KUKA KRL program: demo_posicionaCubos.src, demo_posicionaCubos.dat

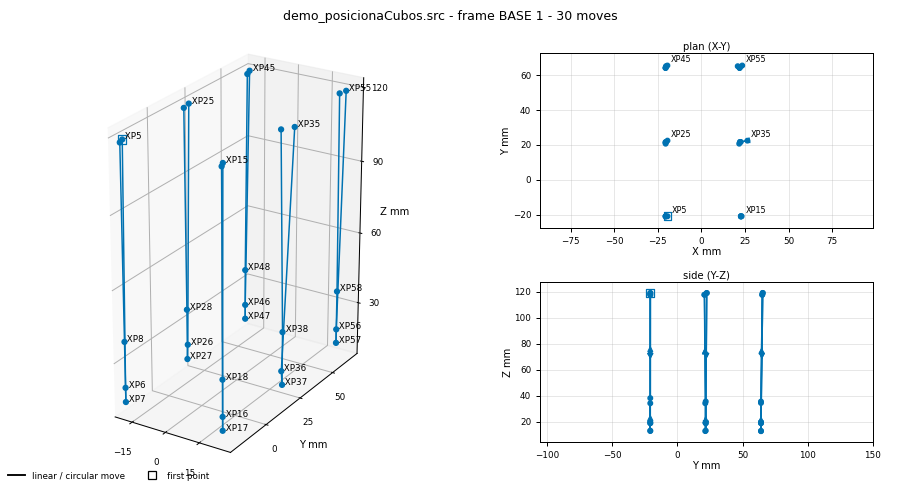
[picture p0: tool path of demo_posicionaCubos.src in frame BASE 1, 30 of 61 moves have a stored position in this frame; points joined in program order, loops and branches not executed]
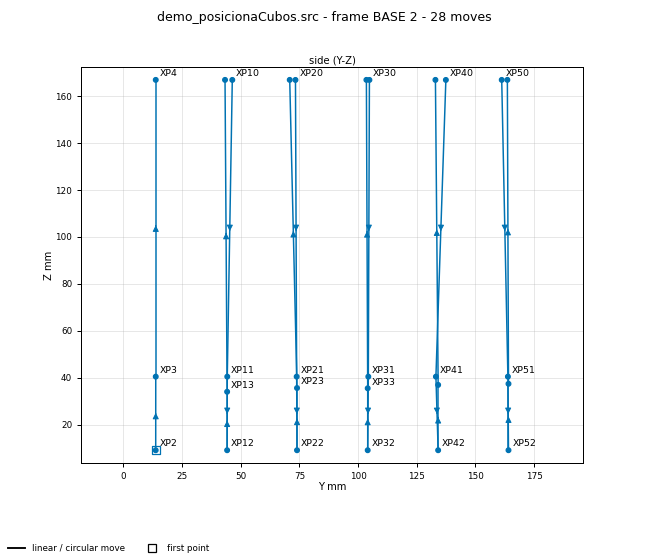
[picture p1: tool path of demo_posicionaCubos.src in frame BASE 2, 28 of 61 moves have a stored position in this frame; points joined in program order, loops and branches not executed]
--- demo_posicionaCubos.src ---
&ACCESS RVO1
&REL 186
&PARAM EDITMASK = *
&PARAM TEMPLATE = C:\KRC\Roboter\Template\vorgabe
DEF demo_posicionaCubos( )
;FOLD INI;%{PE}
  ;FOLD BASISTECH INI
    GLOBAL INTERRUPT DECL 3 WHEN $STOPMESS==TRUE DO IR_STOPM ( )
    INTERRUPT ON 3
    BAS (#INITMOV,0 )
  ;ENDFOLD (BASISTECH INI)
;FOLD SPOTTECH INI
USERSPOT(#INIT)
;ENDFOLD (SPOTTECH INI)
;FOLD GRIPPERTECH INI
USER_GRP(0,DUMMY,DUMMY,GDEFAULT)
;ENDFOLD (GRIPPERTECH INI)
  ;FOLD USER INI
    ;Make your modifications here

  ;ENDFOLD (USER INI)
;ENDFOLD (INI)
;FOLD SET GRIPPER_DEFAULT State=OPN CONT at START Delay=0 ms;%{PE}%R 8.3.1,%MKUKATPGRP,%CGRP,%VGRP,%P 2:1, 4:1, 5:#YES, 6:GDAT0, 8:0, 10:0
TRIGGER WHEN DISTANCE=0 DELAY=0 DO H50(GRP_APO,1,1,GCONT) PRIO=-1
;ENDFOLD
;FOLD PTP HOME  Vel= 100 % DEFAULT;%{PE}%MKUKATPBASIS,%CMOVE,%VPTP,%P 1:PTP, 2:HOME, 3:, 5:100, 7:DEFAULT
$BWDSTART = FALSE
PDAT_ACT=PDEFAULT
FDAT_ACT=FHOME
BAS (#PTP_PARAMS,100 )
$H_POS=XHOME
PTP  XHOME
;ENDFOLD
;FOLD PTP P1 CONT Vel=100 % PDAT2 Tool[1]:Gripper Base[0];%{PE}%R 8.3.34,%MKUKATPBASIS,%CMOVE,%VPTP,%P 1:PTP, 2:P1, 3:C_DIS, 5:100, 7:PDAT2
$BWDSTART=FALSE
PDAT_ACT=PPDAT2
FDAT_ACT=FP1
BAS(#PTP_PARAMS,100)
PTP XP1 C_DIS
;ENDFOLD
;FOLD LIN P2 CONT Vel=0.2 m/s CPDAT53 Tool[1]:Gripper Base[2]:cube_holder;%{PE}%R 8.3.34,%MKUKATPBASIS,%CMOVE,%VLIN,%P 1:LIN, 2:P2, 3:C_DIS C_DIS, 5:0.2, 7:CPDAT53
$BWDSTART=FALSE
LDAT_ACT=LCPDAT53
FDAT_ACT=FP2
BAS(#CP_PARAMS,0.2)
LIN XP2 C_DIS C_DIS
;ENDFOLD
;FOLD SET GRIPPER_DEFAULT State=CLO GDAT1;%{PE}%R 8.3.1,%MKUKATPGRP,%CGRP,%VGRP,%P 2:1, 4:2, 5:#NO, 6:GDAT1, 8:0, 10:0
H50(GRP,1,2,GGDAT1)
;ENDFOLD
;FOLD LIN P3 CONT Vel=0.2 m/s CPDAT54 Tool[1]:Gripper Base[2]:cube_holder;%{PE}%R 8.3.34,%MKUKATPBASIS,%CMOVE,%VLIN,%P 1:LIN, 2:P3, 3:C_DIS C_DIS, 5:0.2, 7:CPDAT54
$BWDSTART=FALSE
LDAT_ACT=LCPDAT54
FDAT_ACT=FP3
BAS(#CP_PARAMS,0.2)
LIN XP3 C_DIS C_DIS
;ENDFOLD
;FOLD LIN P4 CONT Vel=0.5 m/s CPDAT61 Tool[1]:Gripper Base[2]:cube_holder;%{PE}%R 8.3.34,%MKUKATPBASIS,%CMOVE,%VLIN,%P 1:LIN, 2:P4, 3:C_DIS C_DIS, 5:0.5, 7:CPDAT61
$BWDSTART=FALSE
LDAT_ACT=LCPDAT61
FDAT_ACT=FP4
BAS(#CP_PARAMS,0.5)
LIN XP4 C_DIS C_DIS
;ENDFOLD
;FOLD PTP P5 CONT Vel=80 % PDAT18 Tool[1]:Gripper Base[1]:verde;%{PE}%R 8.3.34,%MKUKATPBASIS,%CMOVE,%VPTP,%P 1:PTP, 2:P5, 3:C_DIS, 5:80, 7:PDAT18
$BWDSTART=FALSE
PDAT_ACT=PPDAT18
FDAT_ACT=FP5
BAS(#PTP_PARAMS,80)
PTP XP5 C_DIS
;ENDFOLD
;FOLD LIN P6 CONT Vel=0.5 m/s CPDAT57 Tool[1]:Gripper Base[1]:verde;%{PE}%R 8.3.34,%MKUKATPBASIS,%CMOVE,%VLIN,%P 1:LIN, 2:P6, 3:C_DIS C_DIS, 5:0.5, 7:CPDAT57
$BWDSTART=FALSE
LDAT_ACT=LCPDAT57
FDAT_ACT=FP6
BAS(#CP_PARAMS,0.5)
LIN XP6 C_DIS C_DIS
;ENDFOLD
;FOLD LIN P7 CONT Vel=0.2 m/s CPDAT58 Tool[1]:Gripper Base[1]:verde;%{PE}%R 8.3.34,%MKUKATPBASIS,%CMOVE,%VLIN,%P 1:LIN, 2:P7, 3:C_DIS C_DIS, 5:0.2, 7:CPDAT58
$BWDSTART=FALSE
LDAT_ACT=LCPDAT58
FDAT_ACT=FP7
BAS(#CP_PARAMS,0.2)
LIN XP7 C_DIS C_DIS
;ENDFOLD
;FOLD SET GRIPPER_DEFAULT State=OPN GDAT14;%{PE}%R 8.3.1,%MKUKATPGRP,%CGRP,%VGRP,%P 2:1, 4:1, 5:#NO, 6:GDAT14, 8:0, 10:0
H50(GRP,1,1,GGDAT14)
;ENDFOLD
;FOLD LIN P8 CONT Vel=0.2 m/s CPDAT59 Tool[1]:Gripper Base[1]:verde;%{PE}%R 8.3.34,%MKUKATPBASIS,%CMOVE,%VLIN,%P 1:LIN, 2:P8, 3:C_DIS C_DIS, 5:0.2, 7:CPDAT59
$BWDSTART=FALSE
LDAT_ACT=LCPDAT59
FDAT_ACT=FP8
BAS(#CP_PARAMS,0.2)
LIN XP8 C_DIS C_DIS
;ENDFOLD
;FOLD LIN P9 CONT Vel=0.5 m/s CPDAT60 Tool[1]:Gripper Base[1]:verde;%{PE}%R 8.3.34,%MKUKATPBASIS,%CMOVE,%VLIN,%P 1:LIN, 2:P9, 3:C_DIS C_DIS, 5:0.5, 7:CPDAT60
$BWDSTART=FALSE
LDAT_ACT=LCPDAT60
FDAT_ACT=FP9
BAS(#CP_PARAMS,0.5)
LIN XP9 C_DIS C_DIS
;ENDFOLD
;FOLD PTP P10 CONT Vel=80 % PDAT19 Tool[1]:Gripper Base[2]:cube_holder;%{PE}%R 8.3.34,%MKUKATPBASIS,%CMOVE,%VPTP,%P 1:PTP, 2:P10, 3:C_DIS, 5:80, 7:PDAT19
$BWDSTART=FALSE
PDAT_ACT=PPDAT19
FDAT_ACT=FP10
BAS(#PTP_PARAMS,80)
PTP XP10 C_DIS
;ENDFOLD
;FOLD LIN P11 CONT Vel=0.5 m/s CPDAT62 Tool[1]:Gripper Base[2]:cube_holder;%{PE}%R 8.3.34,%MKUKATPBASIS,%CMOVE,%VLIN,%P 1:LIN, 2:P11, 3:C_DIS C_DIS, 5:0.5, 7:CPDAT62
$BWDSTART=FALSE
LDAT_ACT=LCPDAT62
FDAT_ACT=FP11
BAS(#CP_PARAMS,0.5)
LIN XP11 C_DIS C_DIS
;ENDFOLD
;FOLD LIN P12 CONT Vel=0.2 m/s CPDAT63 Tool[1]:Gripper Base[2]:cube_holder;%{PE}%R 8.3.34,%MKUKATPBASIS,%CMOVE,%VLIN,%P 1:LIN, 2:P12, 3:C_DIS C_DIS, 5:0.2, 7:CPDAT63
$BWDSTART=FALSE
LDAT_ACT=LCPDAT63
FDAT_ACT=FP12
BAS(#CP_PARAMS,0.2)
LIN XP12 C_DIS C_DIS
;ENDFOLD
;FOLD SET GRIPPER_DEFAULT State=CLO GDAT15;%{PE}%R 8.3.1,%MKUKATPGRP,%CGRP,%VGRP,%P 2:1, 4:2, 5:#NO, 6:GDAT15, 8:0, 10:0
H50(GRP,1,2,GGDAT15)
;ENDFOLD
;FOLD LIN P13 CONT Vel=0.2 m/s CPDAT64 Tool[1]:Gripper Base[2]:cube_holder;%{PE}%R 8.3.34,%MKUKATPBASIS,%CMOVE,%VLIN,%P 1:LIN, 2:P13, 3:C_DIS C_DIS, 5:0.2, 7:CPDAT64
$BWDSTART=FALSE
LDAT_ACT=LCPDAT64
FDAT_ACT=FP13
BAS(#CP_PARAMS,0.2)
LIN XP13 C_DIS C_DIS
;ENDFOLD
;FOLD LIN P14 CONT Vel=0.5 m/s CPDAT65 Tool[1]:Gripper Base[2]:cube_holder;%{PE}%R 8.3.34,%MKUKATPBASIS,%CMOVE,%VLIN,%P 1:LIN, 2:P14, 3:C_DIS C_DIS, 5:0.5, 7:CPDAT65
$BWDSTART=FALSE
LDAT_ACT=LCPDAT65
FDAT_ACT=FP14
BAS(#CP_PARAMS,0.5)
LIN XP14 C_DIS C_DIS
;ENDFOLD
;FOLD PTP P15 CONT Vel=80 % PDAT20 Tool[1]:Gripper Base[1]:verde;%{PE}%R 8.3.34,%MKUKATPBASIS,%CMOVE,%VPTP,%P 1:PTP, 2:P15, 3:C_DIS, 5:80, 7:PDAT20
$BWDSTART=FALSE
PDAT_ACT=PPDAT20
FDAT_ACT=FP15
BAS(#PTP_PARAMS,80)
PTP XP15 C_DIS
;ENDFOLD
;FOLD LIN P16 CONT Vel=0.5 m/s CPDAT66 Tool[1]:Gripper Base[1]:verde;%{PE}%R 8.3.34,%MKUKATPBASIS,%CMOVE,%VLIN,%P 1:LIN, 2:P16, 3:C_DIS C_DIS, 5:0.5, 7:CPDAT66
$BWDSTART=FALSE
LDAT_ACT=LCPDAT66
FDAT_ACT=FP16
BAS(#CP_PARAMS,0.5)
LIN XP16 C_DIS C_DIS
;ENDFOLD
;FOLD LIN P17 CONT Vel=0.2 m/s CPDAT67 Tool[1]:Gripper Base[1]:verde;%{PE}%R 8.3.34,%MKUKATPBASIS,%CMOVE,%VLIN,%P 1:LIN, 2:P17, 3:C_DIS C_DIS, 5:0.2, 7:CPDAT67
$BWDSTART=FALSE
LDAT_ACT=LCPDAT67
FDAT_ACT=FP17
BAS(#CP_PARAMS,0.2)
LIN XP17 C_DIS C_DIS
;ENDFOLD
;FOLD SET GRIPPER_DEFAULT State=OPN GDAT16;%{PE}%R 8.3.1,%MKUKATPGRP,%CGRP,%VGRP,%P 2:1, 4:1, 5:#NO, 6:GDAT16, 8:0, 10:0
H50(GRP,1,1,GGDAT16)
;ENDFOLD
;FOLD LIN P18 CONT Vel=0.2 m/s CPDAT69 Tool[1]:Gripper Base[1]:verde;%{PE}%R 8.3.34,%MKUKATPBASIS,%CMOVE,%VLIN,%P 1:LIN, 2:P18, 3:C_DIS C_DIS, 5:0.2, 7:CPDAT69
$BWDSTART=FALSE
LDAT_ACT=LCPDAT69
FDAT_ACT=FP18
BAS(#CP_PARAMS,0.2)
LIN XP18 C_DIS C_DIS
;ENDFOLD
;FOLD LIN P19 CONT Vel=0.5 m/s CPDAT70 Tool[1]:Gripper Base[1]:verde;%{PE}%R 8.3.34,%MKUKATPBASIS,%CMOVE,%VLIN,%P 1:LIN, 2:P19, 3:C_DIS C_DIS, 5:0.5, 7:CPDAT70
$BWDSTART=FALSE
LDAT_ACT=LCPDAT70
FDAT_ACT=FP19
BAS(#CP_PARAMS,0.5)
LIN XP19 C_DIS C_DIS
;ENDFOLD
;FOLD PTP P20 CONT Vel=80 % PDAT21 Tool[1]:Gripper Base[2]:cube_holder;%{PE}%R 8.3.34,%MKUKATPBASIS,%CMOVE,%VPTP,%P 1:PTP, 2:P20, 3:C_DIS, 5:80, 7:PDAT21
$BWDSTART=FALSE
PDAT_ACT=PPDAT21
FDAT_ACT=FP20
BAS(#PTP_PARAMS,80)
PTP XP20 C_DIS
;ENDFOLD
;FOLD LIN P21 CONT Vel=0.5 m/s CPDAT71 Tool[1]:Gripper Base[2]:cube_holder;%{PE}%R 8.3.34,%MKUKATPBASIS,%CMOVE,%VLIN,%P 1:LIN, 2:P21, 3:C_DIS C_DIS, 5:0.5, 7:CPDAT71
$BWDSTART=FALSE
LDAT_ACT=LCPDAT71
FDAT_ACT=FP21
BAS(#CP_PARAMS,0.5)
LIN XP21 C_DIS C_DIS
;ENDFOLD
;FOLD LIN P22 CONT Vel=0.2 m/s CPDAT72 Tool[1]:Gripper Base[2]:cube_holder;%{PE}%R 8.3.34,%MKUKATPBASIS,%CMOVE,%VLIN,%P 1:LIN, 2:P22, 3:C_DIS C_DIS, 5:0.2, 7:CPDAT72
$BWDSTART=FALSE
LDAT_ACT=LCPDAT72
FDAT_ACT=FP22
BAS(#CP_PARAMS,0.2)
LIN XP22 C_DIS C_DIS
;ENDFOLD
;FOLD SET GRIPPER_DEFAULT State=CLO GDAT17;%{PE}%R 8.3.1,%MKUKATPGRP,%CGRP,%VGRP,%P 2:1, 4:2, 5:#NO, 6:GDAT17, 8:0, 10:0
H50(GRP,1,2,GGDAT17)
;ENDFOLD
;FOLD LIN P23 CONT Vel=0.2 m/s CPDAT73 Tool[1]:Gripper Base[2]:cube_holder;%{PE}%R 8.3.34,%MKUKATPBASIS,%CMOVE,%VLIN,%P 1:LIN, 2:P23, 3:C_DIS C_DIS, 5:0.2, 7:CPDAT73
$BWDSTART=FALSE
LDAT_ACT=LCPDAT73
FDAT_ACT=FP23
BAS(#CP_PARAMS,0.2)
LIN XP23 C_DIS C_DIS
;ENDFOLD
;FOLD LIN P24 CONT Vel=0.5 m/s CPDAT74 Tool[1]:Gripper Base[2]:cube_holder;%{PE}%R 8.3.34,%MKUKATPBASIS,%CMOVE,%VLIN,%P 1:LIN, 2:P24, 3:C_DIS C_DIS, 5:0.5, 7:CPDAT74
$BWDSTART=FALSE
LDAT_ACT=LCPDAT74
FDAT_ACT=FP24
BAS(#CP_PARAMS,0.5)
LIN XP24 C_DIS C_DIS
;ENDFOLD
;FOLD PTP P25 CONT Vel=80 % PDAT22 Tool[1]:Gripper Base[1]:verde;%{PE}%R 8.3.34,%MKUKATPBASIS,%CMOVE,%VPTP,%P 1:PTP, 2:P25, 3:C_DIS, 5:80, 7:PDAT22
$BWDSTART=FALSE
PDAT_ACT=PPDAT22
FDAT_ACT=FP25
BAS(#PTP_PARAMS,80)
PTP XP25 C_DIS
;ENDFOLD
;FOLD LIN P26 CONT Vel=0.5 m/s CPDAT75 Tool[1]:Gripper Base[1]:verde;%{PE}%R 8.3.34,%MKUKATPBASIS,%CMOVE,%VLIN,%P 1:LIN, 2:P26, 3:C_DIS C_DIS, 5:0.5, 7:CPDAT75
$BWDSTART=FALSE
LDAT_ACT=LCPDAT75
FDAT_ACT=FP26
BAS(#CP_PARAMS,0.5)
LIN XP26 C_DIS C_DIS
;ENDFOLD
;FOLD LIN P27 CONT Vel=0.2 m/s CPDAT76 Tool[1]:Gripper Base[1]:verde;%{PE}%R 8.3.34,%MKUKATPBASIS,%CMOVE,%VLIN,%P 1:LIN, 2:P27, 3:C_DIS C_DIS, 5:0.2, 7:CPDAT76
$BWDSTART=FALSE
LDAT_ACT=LCPDAT76
FDAT_ACT=FP27
BAS(#CP_PARAMS,0.2)
LIN XP27 C_DIS C_DIS
;ENDFOLD
;FOLD SET GRIPPER_DEFAULT State=OPN GDAT18;%{PE}%R 8.3.1,%MKUKATPGRP,%CGRP,%VGRP,%P 2:1, 4:1, 5:#NO, 6:GDAT18, 8:0, 10:0
H50(GRP,1,1,GGDAT18)
;ENDFOLD
;FOLD LIN P28 CONT Vel=0.2 m/s CPDAT77 Tool[1]:Gripper Base[1]:verde;%{PE}%R 8.3.34,%MKUKATPBASIS,%CMOVE,%VLIN,%P 1:LIN, 2:P28, 3:C_DIS C_DIS, 5:0.2, 7:CPDAT77
$BWDSTART=FALSE
LDAT_ACT=LCPDAT77
FDAT_ACT=FP28
BAS(#CP_PARAMS,0.2)
LIN XP28 C_DIS C_DIS
;ENDFOLD
;FOLD LIN P29 CONT Vel=0.5 m/s CPDAT78 Tool[1]:Gripper Base[1]:verde;%{PE}%R 8.3.34,%MKUKATPBASIS,%CMOVE,%VLIN,%P 1:LIN, 2:P29, 3:C_DIS C_DIS, 5:0.5, 7:CPDAT78
$BWDSTART=FALSE
LDAT_ACT=LCPDAT78
FDAT_ACT=FP29
BAS(#CP_PARAMS,0.5)
LIN XP29 C_DIS C_DIS
;ENDFOLD
;FOLD PTP P30 CONT Vel=80 % PDAT23 Tool[1]:Gripper Base[2]:cube_holder;%{PE}%R 8.3.34,%MKUKATPBASIS,%CMOVE,%VPTP,%P 1:PTP, 2:P30, 3:C_DIS, 5:80, 7:PDAT23
$BWDSTART=FALSE
PDAT_ACT=PPDAT23
FDAT_ACT=FP30
BAS(#PTP_PARAMS,80)
PTP XP30 C_DIS
;ENDFOLD
;FOLD LIN P31 CONT Vel=0.5 m/s CPDAT79 Tool[1]:Gripper Base[2]:cube_holder;%{PE}%R 8.3.34,%MKUKATPBASIS,%CMOVE,%VLIN,%P 1:LIN, 2:P31, 3:C_DIS C_DIS, 5:0.5, 7:CPDAT79
$BWDSTART=FALSE
LDAT_ACT=LCPDAT79
FDAT_ACT=FP31
BAS(#CP_PARAMS,0.5)
LIN XP31 C_DIS C_DIS
;ENDFOLD
;FOLD LIN P32 CONT Vel=0.2 m/s CPDAT80 Tool[1]:Gripper Base[2]:cube_holder;%{PE}%R 8.3.34,%MKUKATPBASIS,%CMOVE,%VLIN,%P 1:LIN, 2:P32, 3:C_DIS C_DIS, 5:0.2, 7:CPDAT80
$BWDSTART=FALSE
LDAT_ACT=LCPDAT80
FDAT_ACT=FP32
BAS(#CP_PARAMS,0.2)
LIN XP32 C_DIS C_DIS
;ENDFOLD
;FOLD SET GRIPPER_DEFAULT State=CLO GDAT19;%{PE}%R 8.3.1,%MKUKATPGRP,%CGRP,%VGRP,%P 2:1, 4:2, 5:#NO, 6:GDAT19, 8:0, 10:0
H50(GRP,1,2,GGDAT19)
;ENDFOLD
;FOLD LIN P33 CONT Vel=0.2 m/s CPDAT81 Tool[1]:Gripper Base[2]:cube_holder;%{PE}%R 8.3.34,%MKUKATPBASIS,%CMOVE,%VLIN,%P 1:LIN, 2:P33, 3:C_DIS C_DIS, 5:0.2, 7:CPDAT81
$BWDSTART=FALSE
LDAT_ACT=LCPDAT81
FDAT_ACT=FP33
BAS(#CP_PARAMS,0.2)
LIN XP33 C_DIS C_DIS
;ENDFOLD
;FOLD LIN P34 CONT Vel=0.5 m/s CPDAT82 Tool[1]:Gripper Base[2]:cube_holder;%{PE}%R 8.3.34,%MKUKATPBASIS,%CMOVE,%VLIN,%P 1:LIN, 2:P34, 3:C_DIS C_DIS, 5:0.5, 7:CPDAT82
$BWDSTART=FALSE
LDAT_ACT=LCPDAT82
FDAT_ACT=FP34
BAS(#CP_PARAMS,0.5)
LIN XP34 C_DIS C_DIS
;ENDFOLD
;FOLD PTP P35 CONT Vel=80 % PDAT24 Tool[1]:Gripper Base[1]:verde;%{PE}%R 8.3.34,%MKUKATPBASIS,%CMOVE,%VPTP,%P 1:PTP, 2:P35, 3:C_DIS, 5:80, 7:PDAT24
$BWDSTART=FALSE
PDAT_ACT=PPDAT24
FDAT_ACT=FP35
BAS(#PTP_PARAMS,80)
PTP XP35 C_DIS
;ENDFOLD
;FOLD LIN P36 CONT Vel=0.5 m/s CPDAT83 Tool[1]:Gripper Base[1]:verde;%{PE}%R 8.3.34,%MKUKATPBASIS,%CMOVE,%VLIN,%P 1:LIN, 2:P36, 3:C_DIS C_DIS, 5:0.5, 7:CPDAT83
$BWDSTART=FALSE
LDAT_ACT=LCPDAT83
FDAT_ACT=FP36
BAS(#CP_PARAMS,0.5)
LIN XP36 C_DIS C_DIS
;ENDFOLD
;FOLD LIN P37 CONT Vel=0.2 m/s CPDAT84 Tool[1]:Gripper Base[1]:verde;%{PE}%R 8.3.34,%MKUKATPBASIS,%CMOVE,%VLIN,%P 1:LIN, 2:P37, 3:C_DIS C_DIS, 5:0.2, 7:CPDAT84
$BWDSTART=FALSE
LDAT_ACT=LCPDAT84
FDAT_ACT=FP37
BAS(#CP_PARAMS,0.2)
LIN XP37 C_DIS C_DIS
;ENDFOLD
;FOLD SET GRIPPER_DEFAULT State=OPN GDAT20;%{PE}%R 8.3.1,%MKUKATPGRP,%CGRP,%VGRP,%P 2:1, 4:1, 5:#NO, 6:GDAT20, 8:0, 10:0
H50(GRP,1,1,GGDAT20)
;ENDFOLD
;FOLD LIN P38 CONT Vel=0.2 m/s CPDAT85 Tool[1]:Gripper Base[1]:verde;%{PE}%R 8.3.34,%MKUKATPBASIS,%CMOVE,%VLIN,%P 1:LIN, 2:P38, 3:C_DIS C_DIS, 5:0.2, 7:CPDAT85
$BWDSTART=FALSE
LDAT_ACT=LCPDAT85
FDAT_ACT=FP38
BAS(#CP_PARAMS,0.2)
LIN XP38 C_DIS C_DIS
;ENDFOLD
;FOLD LIN P39 CONT Vel=0.5 m/s CPDAT86 Tool[1]:Gripper Base[1]:verde;%{PE}%R 8.3.34,%MKUKATPBASIS,%CMOVE,%VLIN,%P 1:LIN, 2:P39, 3:C_DIS C_DIS, 5:0.5, 7:CPDAT86
$BWDSTART=FALSE
LDAT_ACT=LCPDAT86
FDAT_ACT=FP39
BAS(#CP_PARAMS,0.5)
LIN XP39 C_DIS C_DIS
;ENDFOLD
;FOLD PTP P40 CONT Vel=80 % PDAT25 Tool[1]:Gripper Base[2]:cube_holder;%{PE}%R 8.3.34,%MKUKATPBASIS,%CMOVE,%VPTP,%P 1:PTP, 2:P40, 3:C_DIS, 5:80, 7:PDAT25
$BWDSTART=FALSE
PDAT_ACT=PPDAT25
FDAT_ACT=FP40
BAS(#PTP_PARAMS,80)
PTP XP40 C_DIS
;ENDFOLD
;FOLD LIN P41 CONT Vel=0.5 m/s CPDAT87 Tool[1]:Gripper Base[2]:cube_holder;%{PE}%R 8.3.34,%MKUKATPBASIS,%CMOVE,%VLIN,%P 1:LIN, 2:P41, 3:C_DIS C_DIS, 5:0.5, 7:CPDAT87
$BWDSTART=FALSE
LDAT_ACT=LCPDAT87
FDAT_ACT=FP41
BAS(#CP_PARAMS,0.5)
LIN XP41 C_DIS C_DIS
;ENDFOLD
;FOLD LIN P42 CONT Vel=0.2 m/s CPDAT88 Tool[1]:Gripper Base[2]:cube_holder;%{PE}%R 8.3.34,%MKUKATPBASIS,%CMOVE,%VLIN,%P 1:LIN, 2:P42, 3:C_DIS C_DIS, 5:0.2, 7:CPDAT88
$BWDSTART=FALSE
LDAT_ACT=LCPDAT88
FDAT_ACT=FP42
BAS(#CP_PARAMS,0.2)
LIN XP42 C_DIS C_DIS
;ENDFOLD
;FOLD SET GRIPPER_DEFAULT State=CLO GDAT21;%{PE}%R 8.3.1,%MKUKATPGRP,%CGRP,%VGRP,%P 2:1, 4:2, 5:#NO, 6:GDAT21, 8:0, 10:0
H50(GRP,1,2,GGDAT21)
;ENDFOLD
;FOLD LIN P43 CONT Vel=0.2 m/s CPDAT89 Tool[1]:Gripper Base[2]:cube_holder;%{PE}%R 8.3.34,%MKUKATPBASIS,%CMOVE,%VLIN,%P 1:LIN, 2:P43, 3:C_DIS C_DIS, 5:0.2, 7:CPDAT89
$BWDSTART=FALSE
LDAT_ACT=LCPDAT89
FDAT_ACT=FP43
BAS(#CP_PARAMS,0.2)
LIN XP43 C_DIS C_DIS
;ENDFOLD
;FOLD LIN P44 CONT Vel=0.5 m/s CPDAT90 Tool[1]:Gripper Base[2]:cube_holder;%{PE}%R 8.3.34,%MKUKATPBASIS,%CMOVE,%VLIN,%P 1:LIN, 2:P44, 3:C_DIS C_DIS, 5:0.5, 7:CPDAT90
$BWDSTART=FALSE
LDAT_ACT=LCPDAT90
FDAT_ACT=FP44
BAS(#CP_PARAMS,0.5)
LIN XP44 C_DIS C_DIS
;ENDFOLD
;FOLD PTP P45 CONT Vel=80 % PDAT26 Tool[1]:Gripper Base[1]:verde;%{PE}%R 8.3.34,%MKUKATPBASIS,%CMOVE,%VPTP,%P 1:PTP, 2:P45, 3:C_DIS, 5:80, 7:PDAT26
$BWDSTART=FALSE
PDAT_ACT=PPDAT26
FDAT_ACT=FP45
BAS(#PTP_PARAMS,80)
PTP XP45 C_DIS
;ENDFOLD
;FOLD LIN P46 CONT Vel=0.5 m/s CPDAT91 Tool[1]:Gripper Base[1]:verde;%{PE}%R 8.3.34,%MKUKATPBASIS,%CMOVE,%VLIN,%P 1:LIN, 2:P46, 3:C_DIS C_DIS, 5:0.5, 7:CPDAT91
$BWDSTART=FALSE
LDAT_ACT=LCPDAT91
FDAT_ACT=FP46
BAS(#CP_PARAMS,0.5)
LIN XP46 C_DIS C_DIS
;ENDFOLD
;FOLD LIN P47 CONT Vel=0.2 m/s CPDAT92 Tool[1]:Gripper Base[1]:verde;%{PE}%R 8.3.34,%MKUKATPBASIS,%CMOVE,%VLIN,%P 1:LIN, 2:P47, 3:C_DIS C_DIS, 5:0.2, 7:CPDAT92
$BWDSTART=FALSE
LDAT_ACT=LCPDAT92
FDAT_ACT=FP47
BAS(#CP_PARAMS,0.2)
LIN XP47 C_DIS C_DIS
;ENDFOLD
;FOLD SET GRIPPER_DEFAULT State=OPN GDAT22;%{PE}%R 8.3.1,%MKUKATPGRP,%CGRP,%VGRP,%P 2:1, 4:1, 5:#NO, 6:GDAT22, 8:0, 10:0
H50(GRP,1,1,GGDAT22)
;ENDFOLD
;FOLD LIN P48 CONT Vel=0.2 m/s CPDAT93 Tool[1]:Gripper Base[1]:verde;%{PE}%R 8.3.34,%MKUKATPBASIS,%CMOVE,%VLIN,%P 1:LIN, 2:P48, 3:C_DIS C_DIS, 5:0.2, 7:CPDAT93
$BWDSTART=FALSE
LDAT_ACT=LCPDAT93
FDAT_ACT=FP48
BAS(#CP_PARAMS,0.2)
LIN XP48 C_DIS C_DIS
;ENDFOLD
;FOLD LIN P49 CONT Vel=0.5 m/s CPDAT94 Tool[1]:Gripper Base[1]:verde;%{PE}%R 8.3.34,%MKUKATPBASIS,%CMOVE,%VLIN,%P 1:LIN, 2:P49, 3:C_DIS C_DIS, 5:0.5, 7:CPDAT94
$BWDSTART=FALSE
LDAT_ACT=LCPDAT94
FDAT_ACT=FP49
BAS(#CP_PARAMS,0.5)
LIN XP49 C_DIS C_DIS
;ENDFOLD
;FOLD PTP P50 CONT Vel=80 % PDAT27 Tool[1]:Gripper Base[2]:cube_holder;%{PE}%R 8.3.34,%MKUKATPBASIS,%CMOVE,%VPTP,%P 1:PTP, 2:P50, 3:C_DIS, 5:80, 7:PDAT27
$BWDSTART=FALSE
PDAT_ACT=PPDAT27
FDAT_ACT=FP50
BAS(#PTP_PARAMS,80)
PTP XP50 C_DIS
;ENDFOLD
;FOLD LIN P51 CONT Vel=0.5 m/s CPDAT95 Tool[1]:Gripper Base[2]:cube_holder;%{PE}%R 8.3.34,%MKUKATPBASIS,%CMOVE,%VLIN,%P 1:LIN, 2:P51, 3:C_DIS C_DIS, 5:0.5, 7:CPDAT95
$BWDSTART=FALSE
LDAT_ACT=LCPDAT95
FDAT_ACT=FP51
BAS(#CP_PARAMS,0.5)
LIN XP51 C_DIS C_DIS
;ENDFOLD
;FOLD LIN P52 CONT Vel=0.2 m/s CPDAT96 Tool[1]:Gripper Base[2]:cube_holder;%{PE}%R 8.3.34,%MKUKATPBASIS,%CMOVE,%VLIN,%P 1:LIN, 2:P52, 3:C_DIS C_DIS, 5:0.2, 7:CPDAT96
$BWDSTART=FALSE
LDAT_ACT=LCPDAT96
FDAT_ACT=FP52
BAS(#CP_PARAMS,0.2)
LIN XP52 C_DIS C_DIS
;ENDFOLD
;FOLD SET GRIPPER_DEFAULT State=CLO GDAT23;%{PE}%R 8.3.1,%MKUKATPGRP,%CGRP,%VGRP,%P 2:1, 4:2, 5:#NO, 6:GDAT23, 8:0, 10:0
H50(GRP,1,2,GGDAT23)
;ENDFOLD
;FOLD LIN P53 CONT Vel=0.2 m/s CPDAT97 Tool[1]:Gripper Base[2]:cube_holder;%{PE}%R 8.3.34,%MKUKATPBASIS,%CMOVE,%VLIN,%P 1:LIN, 2:P53, 3:C_DIS C_DIS, 5:0.2, 7:CPDAT97
$BWDSTART=FALSE
LDAT_ACT=LCPDAT97
FDAT_ACT=FP53
BAS(#CP_PARAMS,0.2)
LIN XP53 C_DIS C_DIS
;ENDFOLD
;FOLD LIN P54 CONT Vel=0.5 m/s CPDAT98 Tool[1]:Gripper Base[2]:cube_holder;%{PE}%R 8.3.34,%MKUKATPBASIS,%CMOVE,%VLIN,%P 1:LIN, 2:P54, 3:C_DIS C_DIS, 5:0.5, 7:CPDAT98
$BWDSTART=FALSE
LDAT_ACT=LCPDAT98
FDAT_ACT=FP54
BAS(#CP_PARAMS,0.5)
LIN XP54 C_DIS C_DIS
;ENDFOLD
;FOLD PTP P55 CONT Vel=80 % PDAT28 Tool[1]:Gripper Base[1]:verde;%{PE}%R 8.3.34,%MKUKATPBASIS,%CMOVE,%VPTP,%P 1:PTP, 2:P55, 3:C_DIS, 5:80, 7:PDAT28
$BWDSTART=FALSE
PDAT_ACT=PPDAT28
FDAT_ACT=FP55
BAS(#PTP_PARAMS,80)
PTP XP55 C_DIS
;ENDFOLD
;FOLD LIN P56 CONT Vel=0.5 m/s CPDAT99 Tool[1]:Gripper Base[1]:verde;%{PE}%R 8.3.34,%MKUKATPBASIS,%CMOVE,%VLIN,%P 1:LIN, 2:P56, 3:C_DIS C_DIS, 5:0.5, 7:CPDAT99
$BWDSTART=FALSE
LDAT_ACT=LCPDAT99
FDAT_ACT=FP56
BAS(#CP_PARAMS,0.5)
LIN XP56 C_DIS C_DIS
;ENDFOLD
;FOLD LIN P57 CONT Vel=0.2 m/s CPDAT100 Tool[1]:Gripper Base[1]:verde;%{PE}%R 8.3.34,%MKUKATPBASIS,%CMOVE,%VLIN,%P 1:LIN, 2:P57, 3:C_DIS C_DIS, 5:0.2, 7:CPDAT100
$BWDSTART=FALSE
LDAT_ACT=LCPDAT100
FDAT_ACT=FP57
BAS(#CP_PARAMS,0.2)
LIN XP57 C_DIS C_DIS
;ENDFOLD
;FOLD SET GRIPPER_DEFAULT State=OPN GDAT24;%{PE}%R 8.3.1,%MKUKATPGRP,%CGRP,%VGRP,%P 2:1, 4:1, 5:#NO, 6:GDAT24, 8:0, 10:0
H50(GRP,1,1,GGDAT24)
;ENDFOLD
;FOLD LIN P58 CONT Vel=0.2 m/s CPDAT101 Tool[1]:Gripper Base[1]:verde;%{PE}%R 8.3.34,%MKUKATPBASIS,%CMOVE,%VLIN,%P 1:LIN, 2:P58, 3:C_DIS C_DIS, 5:0.2, 7:CPDAT101
$BWDSTART=FALSE
LDAT_ACT=LCPDAT101
FDAT_ACT=FP58
BAS(#CP_PARAMS,0.2)
LIN XP58 C_DIS C_DIS
;ENDFOLD
;FOLD LIN P59 CONT Vel=0.5 m/s CPDAT102 Tool[1]:Gripper Base[1]:verde;%{PE}%R 8.3.34,%MKUKATPBASIS,%CMOVE,%VLIN,%P 1:LIN, 2:P59, 3:C_DIS C_DIS, 5:0.5, 7:CPDAT102
$BWDSTART=FALSE
LDAT_ACT=LCPDAT102
FDAT_ACT=FP59
BAS(#CP_PARAMS,0.5)
LIN XP59 C_DIS C_DIS
;ENDFOLD
;FOLD PTP HOME Vel=100 % DEFAULT;%{PE}%R 8.3.34,%MKUKATPBASIS,%CMOVE,%VPTP,%P 1:PTP, 2:HOME, 3:, 5:100, 7:DEFAULT
$BWDSTART=FALSE
PDAT_ACT=PDEFAULT
FDAT_ACT=FHOME
BAS(#PTP_PARAMS,100)
$H_POS=XHOME
PTP XHOME
;ENDFOLD
END

--- demo_posicionaCubos.dat ---
&ACCESS RVO1
&REL 186
&PARAM EDITMASK = *
&PARAM TEMPLATE = C:\KRC\Roboter\Template\vorgabe
DEFDAT demo_posicionaCubos
;FOLD EXTERNAL DECLARATIONS;%{PE}%MKUKATPBASIS,%CEXT,%VCOMMON,%P
;FOLD GRIPPERTECH EXT
EXT  H50 (INT  :IN,INT  :IN,INT  :IN,GRP_TYP  :IN )
;ENDFOLD (GRIPPERTECH EXT)
;FOLD SPOTTECH EXT
EXT  USERSPOT (S_COMMAND  :IN,SPOT_TYPE  :IN )
;ENDFOLD (SPOTTECH EXT)
;FOLD BASISTECH EXT;%{PE}%MKUKATPBASIS,%CEXT,%VEXT,%P
EXT  BAS (BAS_COMMAND  :IN,REAL  :IN )
DECL INT SUCCESS
;ENDFOLD (BASISTECH EXT)
;FOLD USER EXT;%{E}%MKUKATPUSER,%CEXT,%VEXT,%P
;Make your modifications here

;ENDFOLD (USER EXT)
;ENDFOLD (EXTERNAL DECLARATIONS)
DECL BASIS_SUGG_T LAST_BASIS={POINT1[] "P129                    ",POINT2[] "P129                    ",CP_PARAMS[] "CPDAT102                ",PTP_PARAMS[] "PDAT28                  ",CONT[] "C_DIS C_DIS             ",CP_VEL[] "0.5                     ",PTP_VEL[] "80                      ",SYNC_PARAMS[] "SYNCDAT                 ",SPL_NAME[] "S0                      ",A_PARAMS[] "ADAT0                   "}
;DECL E6POS XP1={X 596.599182,Y 0.393850207,Z 140.365234,A 89.9984894,B -0.000798609108,C 179.994583,S 2,T 43,E1 0.0,E2 0.0,E3 0.0,E4 0.0,E5 0.0,E6 0.0}
;DECL FDAT FP1={TOOL_NO 1,BASE_NO 0,IPO_FRAME #BASE,POINT2[] " ",TQ_STATE FALSE}
DECL PDAT PPDAT1={VEL 100.000,ACC 30.0000,APO_DIST 100.000,APO_MODE #CDIS,GEAR_JERK 50.0000,EXAX_IGN 0}
;DECL E6POS XP2={X 592.660706,Y -76.1390610,Z 89.0645,A 0.302610636,B 0.00510809803,C 179.994476,S 2,T 34,E1 0.0,E2 0.0,E3 0.0,E4 0.0,E5 0.0,E6 0.0}
;DECL FDAT FP2={TOOL_NO 1,BASE_NO 0,IPO_FRAME #BASE,POINT2[] " ",TQ_STATE FALSE}
DECL LDAT LCPDAT1={VEL 2.00000,ACC 30.0000,APO_DIST 100.000,APO_FAC 50.0000,AXIS_VEL 100.000,AXIS_ACC 100.000,ORI_TYP #VAR,CIRC_TYP #BASE,JERK_FAC 50.0000,GEAR_JERK 50.0000,EXAX_IGN 0}
DECL GRP_SUGG_T LAST_GRP={NUMBER[] "1                       ",STATE[] "1                       ",PARAMS[] "GDAT24                  "}
DECL GRP_TYP GGDAT1={G_APO #NO,GRP_TIME 0.700000,CTRL #OFF,DLY 0,DST 1}
DECL E6POS XP1={X 596.599182,Y 0.393849939,Z 140.365234,A 0.152132228,B -0.000798610621,C 179.994583,S 2,T 35,E1 0.0,E2 0.0,E3 0.0,E4 0.0,E5 0.0,E6 0.0}
DECL FDAT FP1={TOOL_NO 1,BASE_NO 0,IPO_FRAME #BASE,POINT2[] " ",TQ_STATE FALSE}
DECL PDAT PPDAT2={VEL 100.000,ACC 30.0000,APO_DIST 250.000,APO_MODE #CDIS,GEAR_JERK 50.0000,EXAX_IGN 0}
;DECL E6POS XP4={X 592.671936,Y -76.1404800,Z 120.425476,A 0.302610695,B 0.00372258225,C 179.994293,S 2,T 34,E1 0.0,E2 0.0,E3 0.0,E4 0.0,E5 0.0,E6 0.0}
;DECL FDAT FP4={TOOL_NO 1,BASE_NO 0,IPO_FRAME #BASE,POINT2[] " ",TQ_STATE FALSE}
DECL LDAT LCPDAT2={VEL 2.00000,ACC 30.0000,APO_DIST 100.000,APO_FAC 50.0000,AXIS_VEL 100.000,AXIS_ACC 100.000,ORI_TYP #VAR,CIRC_TYP #BASE,JERK_FAC 50.0000,GEAR_JERK 50.0000,EXAX_IGN 0}
;DECL E6POS XP5={X 324.194611,Y 306.101685,Z 267.015259,A 0.302610785,B 0.00205069594,C 179.995865,S 2,T 35,E1 0.0,E2 0.0,E3 0.0,E4 0.0,E5 0.0,E6 0.0}
;DECL FDAT FP5={TOOL_NO 1,BASE_NO 0,IPO_FRAME #BASE,POINT2[] " ",TQ_STATE FALSE}
DECL PDAT PPDAT3={VEL 100.000,ACC 30.0000,APO_DIST 100.000,APO_MODE #CDIS,GEAR_JERK 50.0000,EXAX_IGN 0}
;DECL E6POS XP6={X 322.394409,Y 317.214203,Z 168.306381,A 0.302610844,B -0.00158163835,C 179.999359,S 2,T 35,E1 0.0,E2 0.0,E3 0.0,E4 0.0,E5 0.0,E6 0.0}
;DECL FDAT FP6={TOOL_NO 1,BASE_NO 0,IPO_FRAME #BASE,POINT2[] " ",TQ_STATE FALSE}
DECL LDAT LCPDAT3={VEL 2.00000,ACC 30.0000,APO_DIST 100.000,APO_FAC 50.0000,AXIS_VEL 100.000,AXIS_ACC 100.000,ORI_TYP #VAR,CIRC_TYP #BASE,JERK_FAC 50.0000,GEAR_JERK 50.0000,EXAX_IGN 0}
;DECL E6POS XP7={X 322.394409,Y 317.214203,Z 161.041107,A 0.302610904,B -0.00158164906,C 179.999359,S 2,T 35,E1 0.0,E2 0.0,E3 0.0,E4 0.0,E5 0.0,E6 0.0}
;DECL FDAT FP7={TOOL_NO 1,BASE_NO 0,IPO_FRAME #BASE,POINT2[] " ",TQ_STATE FALSE}
DECL LDAT LCPDAT4={VEL 2.00000,ACC 30.0000,APO_DIST 100.000,APO_FAC 50.0000,AXIS_VEL 100.000,AXIS_ACC 100.000,ORI_TYP #VAR,CIRC_TYP #BASE,JERK_FAC 50.0000,GEAR_JERK 50.0000,EXAX_IGN 0}
DECL GRP_TYP GGDAT2={G_APO #NO,GRP_TIME 0.700000,CTRL #OFF,DLY 0,DST 1}
;DECL E6POS XP8={X 322.394409,Y 317.214203,Z 193.261078,A 0.302610904,B -0.00158164476,C 179.999359,S 2,T 35,E1 0.0,E2 0.0,E3 0.0,E4 0.0,E5 0.0,E6 0.0}
;DECL FDAT FP8={TOOL_NO 1,BASE_NO 0,IPO_FRAME #BASE,POINT2[] " ",TQ_STATE FALSE}
DECL LDAT LCPDAT5={VEL 2.00000,ACC 30.0000,APO_DIST 100.000,APO_FAC 50.0000,AXIS_VEL 100.000,AXIS_ACC 100.000,ORI_TYP #VAR,CIRC_TYP #BASE,JERK_FAC 50.0000,GEAR_JERK 50.0000,EXAX_IGN 0}
;DECL E6POS XP9={X 592.543396,Y -0.190673187,Z 282.661377,A 0.302610934,B 0.0125020090,C 179.999405,S 2,T 35,E1 0.0,E2 0.0,E3 0.0,E4 0.0,E5 0.0,E6 0.0}
;DECL FDAT FP9={TOOL_NO 1,BASE_NO 0,IPO_FRAME #BASE,POINT2[] " ",TQ_STATE FALSE}
DECL PDAT PPDAT4={VEL 100.000,ACC 30.0000,APO_DIST 100.000,APO_MODE #CDIS,GEAR_JERK 50.0000,EXAX_IGN 0}
;DECL E6POS XP10={X 591.553528,Y -45.7813225,Z 118.233986,A 0.303232640,B 0.00849394780,C 179.998764,S 2,T 34,E1 0.0,E2 0.0,E3 0.0,E4 0.0,E5 0.0,E6 0.0}
;DECL FDAT FP10={TOOL_NO 1,BASE_NO 0,IPO_FRAME #BASE,POINT2[] " ",TQ_STATE FALSE}
DECL LDAT LCPDAT6={VEL 2.00000,ACC 30.0000,APO_DIST 100.000,APO_FAC 50.0000,AXIS_VEL 100.000,AXIS_ACC 100.000,ORI_TYP #VAR,CIRC_TYP #BASE,JERK_FAC 50.0000,GEAR_JERK 50.0000,EXAX_IGN 0}
;DECL E6POS XP11={X 592.268494,Y -45.9636612,Z 89.0582581,A 0.303232670,B 0.00849390,C 179.998764,S 2,T 34,E1 0.0,E2 0.0,E3 0.0,E4 0.0,E5 0.0,E6 0.0}
;DECL FDAT FP11={TOOL_NO 1,BASE_NO 0,IPO_FRAME #BASE,POINT2[] " ",TQ_STATE FALSE}
DECL LDAT LCPDAT7={VEL 2.00000,ACC 30.0000,APO_DIST 100.000,APO_FAC 50.0000,AXIS_VEL 100.000,AXIS_ACC 100.000,ORI_TYP #VAR,CIRC_TYP #BASE,JERK_FAC 50.0000,GEAR_JERK 50.0000,EXAX_IGN 0}
DECL GRP_TYP GGDAT3={G_APO #NO,GRP_TIME 0.700000,CTRL #OFF,DLY 0,DST 1}
;DECL E6POS XP12={X 592.265564,Y -45.9625473,Z 117.106590,A 0.302383751,B 0.00838480052,C 179.999023,S 2,T 34,E1 0.0,E2 0.0,E3 0.0,E4 0.0,E5 0.0,E6 0.0}
;DECL FDAT FP12={TOOL_NO 1,BASE_NO 0,IPO_FRAME #BASE,POINT2[] " ",TQ_STATE FALSE}
DECL LDAT LCPDAT8={VEL 2.00000,ACC 30.0000,APO_DIST 100.000,APO_FAC 50.0000,AXIS_VEL 100.000,AXIS_ACC 100.000,ORI_TYP #VAR,CIRC_TYP #BASE,JERK_FAC 50.0000,GEAR_JERK 50.0000,EXAX_IGN 0}
;DECL E6POS XP13={X 592.321960,Y -45.9643669,Z 220.340576,A 0.301014274,B -0.00401754770,C 179.998611,S 2,T 34,E1 0.0,E2 0.0,E3 0.0,E4 0.0,E5 0.0,E6 0.0}
;DECL FDAT FP13={TOOL_NO 1,BASE_NO 0,IPO_FRAME #BASE,POINT2[] " ",TQ_STATE FALSE}
DECL LDAT LCPDAT9={VEL 2.00000,ACC 30.0000,APO_DIST 100.000,APO_FAC 50.0000,AXIS_VEL 100.000,AXIS_ACC 100.000,ORI_TYP #VAR,CIRC_TYP #BASE,JERK_FAC 50.0000,GEAR_JERK 50.0000,EXAX_IGN 0}
DECL PDAT PPDAT5={VEL 100.000,ACC 30.0000,APO_DIST 100.000,APO_MODE #CDIS,GEAR_JERK 50.0000,EXAX_IGN 0}
;DECL E6POS XP14={X 323.552765,Y 274.171143,Z 169.258316,A 0.311525762,B -0.00474398816,C 179.999191,S 2,T 35,E1 0.0,E2 0.0,E3 0.0,E4 0.0,E5 0.0,E6 0.0}
;DECL FDAT FP14={TOOL_NO 1,BASE_NO 0,IPO_FRAME #BASE,POINT2[] " ",TQ_STATE FALSE}
DECL LDAT LCPDAT10={VEL 2.00000,ACC 30.0000,APO_DIST 100.000,APO_FAC 50.0000,AXIS_VEL 100.000,AXIS_ACC 100.000,ORI_TYP #VAR,CIRC_TYP #BASE,JERK_FAC 50.0000,GEAR_JERK 50.0000,EXAX_IGN 0}
;DECL E6POS XP15={X 323.552765,Y 274.171143,Z 161.456985,A 0.311525792,B -0.00474398909,C 179.999191,S 2,T 35,E1 0.0,E2 0.0,E3 0.0,E4 0.0,E5 0.0,E6 0.0}
;DECL FDAT FP15={TOOL_NO 1,BASE_NO 0,IPO_FRAME #BASE,POINT2[] " ",TQ_STATE FALSE}
DECL LDAT LCPDAT11={VEL 2.00000,ACC 30.0000,APO_DIST 100.000,APO_FAC 50.0000,AXIS_VEL 100.000,AXIS_ACC 100.000,ORI_TYP #VAR,CIRC_TYP #BASE,JERK_FAC 50.0000,GEAR_JERK 50.0000,EXAX_IGN 0}
DECL GRP_TYP GGDAT4={G_APO #NO,GRP_TIME 0.700000,CTRL #OFF,DLY 0,DST 1}
;DECL E6POS XP16={X 323.585663,Y 274.202454,Z 183.737228,A 0.312368,B -0.00454253936,C 179.998718,S 2,T 35,E1 0.0,E2 0.0,E3 0.0,E4 0.0,E5 0.0,E6 0.0}
;DECL FDAT FP16={TOOL_NO 1,BASE_NO 0,IPO_FRAME #BASE,POINT2[] " ",TQ_STATE FALSE}
DECL LDAT LCPDAT12={VEL 2.00000,ACC 30.0000,APO_DIST 100.000,APO_FAC 50.0000,AXIS_VEL 100.000,AXIS_ACC 100.000,ORI_TYP #VAR,CIRC_TYP #BASE,JERK_FAC 50.0000,GEAR_JERK 50.0000,EXAX_IGN 0}
;DECL E6POS XP17={X 323.691711,Y 274.284546,Z 388.025696,A 0.313318074,B -0.0243321341,C -179.987579,S 2,T 35,E1 0.0,E2 0.0,E3 0.0,E4 0.0,E5 0.0,E6 0.0}
;DECL FDAT FP17={TOOL_NO 1,BASE_NO 0,IPO_FRAME #BASE,POINT2[] " ",TQ_STATE FALSE}
DECL LDAT LCPDAT13={VEL 2.00000,ACC 30.0000,APO_DIST 100.000,APO_FAC 50.0000,AXIS_VEL 100.000,AXIS_ACC 100.000,ORI_TYP #VAR,CIRC_TYP #BASE,JERK_FAC 50.0000,GEAR_JERK 50.0000,EXAX_IGN 0}
;DECL E6POS XP18={X 598.243164,Y -2.81892347,Z 236.926025,A 0.313317686,B -0.0277198255,C -179.987427,S 2,T 42,E1 0.0,E2 0.0,E3 0.0,E4 0.0,E5 0.0,E6 0.0}
;DECL FDAT FP18={TOOL_NO 1,BASE_NO 0,IPO_FRAME #BASE,POINT2[] " ",TQ_STATE FALSE}
DECL PDAT PPDAT6={VEL 100.000,ACC 30.0000,APO_DIST 100.000,APO_MODE #CDIS,GEAR_JERK 50.0000,EXAX_IGN 0}
;DECL E6POS XP19={X 592.134338,Y -16.5870438,Z 114.245804,A 0.313317925,B -0.0323884189,C -179.987473,S 2,T 42,E1 0.0,E2 0.0,E3 0.0,E4 0.0,E5 0.0,E6 0.0}
;DECL FDAT FP19={TOOL_NO 1,BASE_NO 0,IPO_FRAME #BASE,POINT2[] " ",TQ_STATE FALSE}
DECL LDAT LCPDAT14={VEL 2.00000,ACC 30.0000,APO_DIST 100.000,APO_FAC 50.0000,AXIS_VEL 100.000,AXIS_ACC 100.000,ORI_TYP #VAR,CIRC_TYP #BASE,JERK_FAC 50.0000,GEAR_JERK 50.0000,EXAX_IGN 0}
;DECL E6POS XP20={X 592.255310,Y -16.2822685,Z 89.1617203,A 0.313318223,B -0.0323885567,C -179.987473,S 2,T 42,E1 0.0,E2 0.0,E3 0.0,E4 0.0,E5 0.0,E6 0.0}
;DECL FDAT FP20={TOOL_NO 1,BASE_NO 0,IPO_FRAME #BASE,POINT2[] " ",TQ_STATE FALSE}
DECL LDAT LCPDAT15={VEL 2.00000,ACC 30.0000,APO_DIST 100.000,APO_FAC 50.0000,AXIS_VEL 100.000,AXIS_ACC 100.000,ORI_TYP #VAR,CIRC_TYP #BASE,JERK_FAC 50.0000,GEAR_JERK 50.0000,EXAX_IGN 0}
DECL GRP_TYP GGDAT5={G_APO #NO,GRP_TIME 0.700000,CTRL #OFF,DLY 0,DST 1}
;DECL E6POS XP21={X 592.255310,Y -16.2822685,Z 115.415405,A 0.313318253,B -0.0323885679,C -179.987473,S 2,T 42,E1 0.0,E2 0.0,E3 0.0,E4 0.0,E5 0.0,E6 0.0}
;DECL FDAT FP21={TOOL_NO 1,BASE_NO 0,IPO_FRAME #BASE,POINT2[] " ",TQ_STATE FALSE}
DECL LDAT LCPDAT16={VEL 2.00000,ACC 30.0000,APO_DIST 100.000,APO_FAC 50.0000,AXIS_VEL 100.000,AXIS_ACC 100.000,ORI_TYP #VAR,CIRC_TYP #BASE,JERK_FAC 50.0000,GEAR_JERK 50.0000,EXAX_IGN 0}
;DECL E6POS XP22={X 592.062622,Y -16.2803135,Z 172.983368,A 0.317161173,B 0.00332541275,C -179.987534,S 2,T 42,E1 0.0,E2 0.0,E3 0.0,E4 0.0,E5 0.0,E6 0.0}
;DECL FDAT FP22={TOOL_NO 1,BASE_NO 0,IPO_FRAME #BASE,POINT2[] " ",TQ_STATE FALSE}
DECL LDAT LCPDAT17={VEL 2.00000,ACC 30.0000,APO_DIST 100.000,APO_FAC 50.0000,AXIS_VEL 100.000,AXIS_ACC 100.000,ORI_TYP #VAR,CIRC_TYP #BASE,JERK_FAC 50.0000,GEAR_JERK 50.0000,EXAX_IGN 0}
;DECL E6POS XP23={X 366.539307,Y 317.294464,Z 209.892654,A 0.317158610,B -0.0204064101,C -179.969971,S 2,T 43,E1 0.0,E2 0.0,E3 0.0,E4 0.0,E5 0.0,E6 0.0}
;DECL FDAT FP23={TOOL_NO 1,BASE_NO 0,IPO_FRAME #BASE,POINT2[] " ",TQ_STATE FALSE}
DECL PDAT PPDAT7={VEL 100.000,ACC 30.0000,APO_DIST 100.000,APO_MODE #CDIS,GEAR_JERK 50.0000,EXAX_IGN 0}
;DECL E6POS XP24={X 365.627777,Y 317.316071,Z 164.060699,A 0.317158759,B -0.0204065405,C -179.969971,S 2,T 43,E1 0.0,E2 0.0,E3 0.0,E4 0.0,E5 0.0,E6 0.0}
;DECL FDAT FP24={TOOL_NO 1,BASE_NO 0,IPO_FRAME #BASE,POINT2[] " ",TQ_STATE FALSE}
DECL LDAT LCPDAT18={VEL 2.00000,ACC 30.0000,APO_DIST 100.000,APO_FAC 50.0000,AXIS_VEL 100.000,AXIS_ACC 100.000,ORI_TYP #VAR,CIRC_TYP #BASE,JERK_FAC 50.0000,GEAR_JERK 50.0000,EXAX_IGN 0}
;DECL E6POS XP25={X 365.627777,Y 317.316071,Z 161.141129,A 0.317158788,B -0.0204065684,C -179.969971,S 2,T 43,E1 0.0,E2 0.0,E3 0.0,E4 0.0,E5 0.0,E6 0.0}
;DECL FDAT FP25={TOOL_NO 1,BASE_NO 0,IPO_FRAME #BASE,POINT2[] " ",TQ_STATE FALSE}
DECL LDAT LCPDAT19={VEL 2.00000,ACC 30.0000,APO_DIST 100.000,APO_FAC 50.0000,AXIS_VEL 100.000,AXIS_ACC 100.000,ORI_TYP #VAR,CIRC_TYP #BASE,JERK_FAC 50.0000,GEAR_JERK 50.0000,EXAX_IGN 0}
;DECL E6POS XP26={X 365.627777,Y 317.316071,Z 169.712479,A 0.317158818,B -0.0204065870,C -179.969971,S 2,T 43,E1 0.0,E2 0.0,E3 0.0,E4 0.0,E5 0.0,E6 0.0}
;DECL FDAT FP26={TOOL_NO 1,BASE_NO 0,IPO_FRAME #BASE,POINT2[] " ",TQ_STATE FALSE}
DECL LDAT LCPDAT20={VEL 2.00000,ACC 30.0000,APO_DIST 100.000,APO_FAC 50.0000,AXIS_VEL 100.000,AXIS_ACC 100.000,ORI_TYP #VAR,CIRC_TYP #BASE,JERK_FAC 50.0000,GEAR_JERK 50.0000,EXAX_IGN 0}
;DECL E6POS XP27={X 365.627808,Y 317.316071,Z 169.712479,A 89.9977188,B -0.0204065498,C -179.969971,S 2,T 43,E1 0.0,E2 0.0,E3 0.0,E4 0.0,E5 0.0,E6 0.0}
;DECL FDAT FP27={TOOL_NO 1,BASE_NO 0,IPO_FRAME #BASE,POINT2[] " ",TQ_STATE FALSE}
DECL LDAT LCPDAT21={VEL 2.00000,ACC 30.0000,APO_DIST 100.000,APO_FAC 50.0000,AXIS_VEL 100.000,AXIS_ACC 100.000,ORI_TYP #VAR,CIRC_TYP #BASE,JERK_FAC 50.0000,GEAR_JERK 50.0000,EXAX_IGN 0}
;DECL E6POS XP28={X 367.045624,Y 317.316071,Z 161.069092,A 89.9977188,B -0.0204065591,C -179.969971,S 2,T 43,E1 0.0,E2 0.0,E3 0.0,E4 0.0,E5 0.0,E6 0.0}
;DECL FDAT FP28={TOOL_NO 1,BASE_NO 0,IPO_FRAME #BASE,POINT2[] " ",TQ_STATE FALSE}
DECL LDAT LCPDAT22={VEL 2.00000,ACC 30.0000,APO_DIST 100.000,APO_FAC 50.0000,AXIS_VEL 100.000,AXIS_ACC 100.000,ORI_TYP #VAR,CIRC_TYP #BASE,JERK_FAC 50.0000,GEAR_JERK 50.0000,EXAX_IGN 0}
DECL GRP_TYP GGDAT6={G_APO #NO,GRP_TIME 0.700000,CTRL #OFF,DLY 0,DST 1}
;DECL E6POS XP29={X 367.049194,Y 317.319153,Z 187.478943,A 89.9977188,B -0.0207769386,C -179.970398,S 2,T 43,E1 0.0,E2 0.0,E3 0.0,E4 0.0,E5 0.0,E6 0.0}
;DECL FDAT FP29={TOOL_NO 1,BASE_NO 0,IPO_FRAME #BASE,POINT2[] " ",TQ_STATE FALSE}
DECL LDAT LCPDAT23={VEL 2.00000,ACC 30.0000,APO_DIST 100.000,APO_FAC 50.0000,AXIS_VEL 100.000,AXIS_ACC 100.000,ORI_TYP #VAR,CIRC_TYP #BASE,JERK_FAC 50.0000,GEAR_JERK 50.0000,EXAX_IGN 0}
;DECL E6POS XP30={X 587.506470,Y 19.0465736,Z 256.948120,A -0.00400581537,B -0.0202185530,C -179.970413,S 2,T 43,E1 0.0,E2 0.0,E3 0.0,E4 0.0,E5 0.0,E6 0.0}
;DECL FDAT FP30={TOOL_NO 1,BASE_NO 0,IPO_FRAME #BASE,POINT2[] " ",TQ_STATE FALSE}
DECL PDAT PPDAT8={VEL 100.000,ACC 30.0000,APO_DIST 100.000,APO_MODE #CDIS,GEAR_JERK 50.0000,EXAX_IGN 0}
;DECL E6POS XP31={X 592.063843,Y 13.7504120,Z 111.088753,A -0.00400567707,B -0.0221780986,C -179.970352,S 2,T 43,E1 0.0,E2 0.0,E3 0.0,E4 0.0,E5 0.0,E6 0.0}
;DECL FDAT FP31={TOOL_NO 1,BASE_NO 0,IPO_FRAME #BASE,POINT2[] " ",TQ_STATE FALSE}
DECL LDAT LCPDAT24={VEL 2.00000,ACC 30.0000,APO_DIST 100.000,APO_FAC 50.0000,AXIS_VEL 100.000,AXIS_ACC 100.000,ORI_TYP #VAR,CIRC_TYP #BASE,JERK_FAC 50.0000,GEAR_JERK 50.0000,EXAX_IGN 0}
;DECL E6POS XP32={X 592.477173,Y 13.5850983,Z 89.2669220,A 0.386679083,B -0.0228960104,C -179.970337,S 2,T 43,E1 0.0,E2 0.0,E3 0.0,E4 0.0,E5 0.0,E6 0.0}
;DECL FDAT FP32={TOOL_NO 1,BASE_NO 0,IPO_FRAME #BASE,POINT2[] " ",TQ_STATE FALSE}
DECL LDAT LCPDAT25={VEL 2.00000,ACC 30.0000,APO_DIST 100.000,APO_FAC 50.0000,AXIS_VEL 100.000,AXIS_ACC 100.000,ORI_TYP #VAR,CIRC_TYP #BASE,JERK_FAC 50.0000,GEAR_JERK 50.0000,EXAX_IGN 0}
DECL GRP_TYP GGDAT7={G_APO #NO,GRP_TIME 0.700000,CTRL #OFF,DLY 0,DST 1}
;DECL E6POS XP33={X 592.473511,Y 13.5850077,Z 118.810074,A 0.386679113,B -0.0224354174,C -179.970337,S 2,T 43,E1 0.0,E2 0.0,E3 0.0,E4 0.0,E5 0.0,E6 0.0}
;DECL FDAT FP33={TOOL_NO 1,BASE_NO 0,IPO_FRAME #BASE,POINT2[] " ",TQ_STATE FALSE}
DECL LDAT LCPDAT26={VEL 2.00000,ACC 30.0000,APO_DIST 100.000,APO_FAC 50.0000,AXIS_VEL 100.000,AXIS_ACC 100.000,ORI_TYP #VAR,CIRC_TYP #BASE,JERK_FAC 50.0000,GEAR_JERK 50.0000,EXAX_IGN 0}
;DECL E6POS XP34={X 592.473511,Y 13.5850077,Z 224.483093,A 1.17302096,B -0.0224354472,C -179.970337,S 2,T 43,E1 0.0,E2 0.0,E3 0.0,E4 0.0,E5 0.0,E6 0.0}
;DECL FDAT FP34={TOOL_NO 1,BASE_NO 0,IPO_FRAME #BASE,POINT2[] " ",TQ_STATE FALSE}
DECL PDAT PPDAT9={VEL 100.000,ACC 30.0000,APO_DIST 100.000,APO_MODE #CDIS,GEAR_JERK 50.0000,EXAX_IGN 0}
;DECL E6POS XP35={X 409.466766,Y 315.058685,Z 272.305603,A 90.0046387,B -0.0269225519,C -179.973129,S 2,T 43,E1 0.0,E2 0.0,E3 0.0,E4 0.0,E5 0.0,E6 0.0}
;DECL FDAT FP35={TOOL_NO 1,BASE_NO 0,IPO_FRAME #BASE,POINT2[] " ",TQ_STATE FALSE}
DECL PDAT PPDAT10={VEL 100.000,ACC 30.0000,APO_DIST 100.000,APO_MODE #CDIS,GEAR_JERK 50.0000,EXAX_IGN 0}
;DECL E6POS XP36={X 409.463562,Y 315.056213,Z 188.664795,A 90.0046387,B -0.0269218534,C -179.973129,S 2,T 43,E1 0.0,E2 0.0,E3 0.0,E4 0.0,E5 0.0,E6 0.0}
;DECL FDAT FP36={TOOL_NO 1,BASE_NO 0,IPO_FRAME #BASE,POINT2[] " ",TQ_STATE FALSE}
DECL PDAT PPDAT11={VEL 100.000,ACC 30.0000,APO_DIST 100.000,APO_MODE #CDIS,GEAR_JERK 50.0000,EXAX_IGN 0}
;DECL E6POS XP37={X 409.657898,Y 317.877258,Z 164.008362,A 90.0046387,B -0.0278242,C -179.974304,S 2,T 43,E1 0.0,E2 0.0,E3 0.0,E4 0.0,E5 0.0,E6 0.0}
;DECL FDAT FP37={TOOL_NO 1,BASE_NO 0,IPO_FRAME #BASE,POINT2[] " ",TQ_STATE FALSE}
DECL LDAT LCPDAT27={VEL 2.00000,ACC 30.0000,APO_DIST 100.000,APO_FAC 50.0000,AXIS_VEL 100.000,AXIS_ACC 100.000,ORI_TYP #VAR,CIRC_TYP #BASE,JERK_FAC 50.0000,GEAR_JERK 50.0000,EXAX_IGN 0}
;DECL E6POS XP38={X 409.657898,Y 317.877258,Z 160.999985,A 90.0046387,B -0.0278242193,C -179.974304,S 2,T 43,E1 0.0,E2 0.0,E3 0.0,E4 0.0,E5 0.0,E6 0.0}
;DECL FDAT FP38={TOOL_NO 1,BASE_NO 0,IPO_FRAME #BASE,POINT2[] " ",TQ_STATE FALSE}
DECL LDAT LCPDAT28={VEL 2.00000,ACC 30.0000,APO_DIST 100.000,APO_FAC 50.0000,AXIS_VEL 100.000,AXIS_ACC 100.000,ORI_TYP #VAR,CIRC_TYP #BASE,JERK_FAC 50.0000,GEAR_JERK 50.0000,EXAX_IGN 0}
DECL GRP_TYP GGDAT8={G_APO #NO,GRP_TIME 0.700000,CTRL #OFF,DLY 0,DST 1}
;DECL E6POS XP39={X 409.651794,Y 317.872498,Z 188.396835,A 90.0046387,B -0.0272382144,C -179.973541,S 2,T 43,E1 0.0,E2 0.0,E3 0.0,E4 0.0,E5 0.0,E6 0.0}
;DECL FDAT FP39={TOOL_NO 1,BASE_NO 0,IPO_FRAME #BASE,POINT2[] " ",TQ_STATE FALSE}
DECL LDAT LCPDAT29={VEL 2.00000,ACC 30.0000,APO_DIST 100.000,APO_FAC 50.0000,AXIS_VEL 100.000,AXIS_ACC 100.000,ORI_TYP #VAR,CIRC_TYP #BASE,JERK_FAC 50.0000,GEAR_JERK 50.0000,EXAX_IGN 0}
;DECL E6POS XP40={X 409.679657,Y 317.894165,Z 555.788,A 90.0046387,B -0.0314656645,C -179.978989,S 2,T 43,E1 0.0,E2 0.0,E3 0.0,E4 0.0,E5 0.0,E6 0.0}
;DECL FDAT FP40={TOOL_NO 1,BASE_NO 0,IPO_FRAME #BASE,POINT2[] " ",TQ_STATE FALSE}
DECL PDAT PPDAT12={VEL 100.000,ACC 30.0000,APO_DIST 100.000,APO_MODE #CDIS,GEAR_JERK 50.0000,EXAX_IGN 0}
;DECL E6POS XP41={X 591.568542,Y -197.751801,Z 154.909103,A 0.0338774398,B -0.0475413762,C 179.996796,S 2,T 42,E1 0.0,E2 0.0,E3 0.0,E4 0.0,E5 0.0,E6 0.0}
;DECL FDAT FP41={TOOL_NO 1,BASE_NO 0,IPO_FRAME #BASE,POINT2[] " ",TQ_STATE FALSE}
DECL PDAT PPDAT13={VEL 100.000,ACC 30.0000,APO_DIST 100.000,APO_MODE #CDIS,GEAR_JERK 50.0000,EXAX_IGN 0}
;DECL E6POS XP42={X 591.568542,Y -197.751801,Z 154.909103,A 0.0338774398,B -0.0475413762,C 179.996796,S 2,T 42,E1 0.0,E2 0.0,E3 0.0,E4 0.0,E5 0.0,E6 0.0}
;DECL FDAT FP42={TOOL_NO 1,BASE_NO 0,IPO_FRAME #BASE,POINT2[] " ",TQ_STATE FALSE}
DECL PDAT PPDAT14={VEL 100.000,ACC 30.0000,APO_DIST 100.000,APO_MODE #CDIS,GEAR_JERK 50.0000,EXAX_IGN 0}
;DECL E6POS XP43={X 592.100647,Y -79.0928268,Z 103.298447,A 0.0338778123,B -0.0445956774,C 179.996658,S 2,T 42,E1 0.0,E2 0.0,E3 0.0,E4 0.0,E5 0.0,E6 0.0}
;DECL FDAT FP43={TOOL_NO 1,BASE_NO 0,IPO_FRAME #BASE,POINT2[] " ",TQ_STATE FALSE}
DECL LDAT LCPDAT30={VEL 2.00000,ACC 30.0000,APO_DIST 100.000,APO_FAC 50.0000,AXIS_VEL 100.000,AXIS_ACC 100.000,ORI_TYP #VAR,CIRC_TYP #BASE,JERK_FAC 50.0000,GEAR_JERK 50.0000,EXAX_IGN 0}
;DECL E6POS XP44={X 592.116333,Y 22.3131447,Z 89.9599457,A 0.0338781,B -0.0465635844,C 179.996384,S 2,T 35,E1 0.0,E2 0.0,E3 0.0,E4 0.0,E5 0.0,E6 0.0}
;DECL FDAT FP44={TOOL_NO 1,BASE_NO 0,IPO_FRAME #BASE,POINT2[] " ",TQ_STATE FALSE}
DECL LDAT LCPDAT31={VEL 2.00000,ACC 30.0000,APO_DIST 100.000,APO_FAC 50.0000,AXIS_VEL 100.000,AXIS_ACC 100.000,ORI_TYP #VAR,CIRC_TYP #BASE,JERK_FAC 50.0000,GEAR_JERK 50.0000,EXAX_IGN 0}
;DECL E6POS XP45={X 592.394653,Y 43.9387,Z 89.1218643,A 0.0338781141,B -0.0465636849,C 179.996384,S 2,T 35,E1 0.0,E2 0.0,E3 0.0,E4 0.0,E5 0.0,E6 0.0}
;DECL FDAT FP45={TOOL_NO 1,BASE_NO 0,IPO_FRAME #BASE,POINT2[] " ",TQ_STATE FALSE}
DECL LDAT LCPDAT32={VEL 2.00000,ACC 30.0000,APO_DIST 100.000,APO_FAC 50.0000,AXIS_VEL 100.000,AXIS_ACC 100.000,ORI_TYP #VAR,CIRC_TYP #BASE,JERK_FAC 50.0000,GEAR_JERK 50.0000,EXAX_IGN 0}
DECL GRP_TYP GGDAT9={G_APO #NO,GRP_TIME 0.700000,CTRL #OFF,DLY 0,DST 1}
;DECL E6POS XP46={X 592.363831,Y 43.9363556,Z 119.122726,A 0.0338783488,B -0.0426726639,C 179.996094,S 2,T 35,E1 0.0,E2 0.0,E3 0.0,E4 0.0,E5 0.0,E6 0.0}
;DECL FDAT FP46={TOOL_NO 1,BASE_NO 0,IPO_FRAME #BASE,POINT2[] " ",TQ_STATE FALSE}
DECL LDAT LCPDAT33={VEL 2.00000,ACC 30.0000,APO_DIST 100.000,APO_FAC 50.0000,AXIS_VEL 100.000,AXIS_ACC 100.000,ORI_TYP #VAR,CIRC_TYP #BASE,JERK_FAC 50.0000,GEAR_JERK 50.0000,EXAX_IGN 0}
;DECL E6POS XP47={X 592.363831,Y 43.9363556,Z 239.951691,A 0.0338783525,B -0.0426726714,C 179.996094,S 2,T 35,E1 0.0,E2 0.0,E3 0.0,E4 0.0,E5 0.0,E6 0.0}
;DECL FDAT FP47={TOOL_NO 1,BASE_NO 0,IPO_FRAME #BASE,POINT2[] " ",TQ_STATE FALSE}
DECL LDAT LCPDAT34={VEL 2.00000,ACC 30.0000,APO_DIST 100.000,APO_FAC 50.0000,AXIS_VEL 100.000,AXIS_ACC 100.000,ORI_TYP #VAR,CIRC_TYP #BASE,JERK_FAC 50.0000,GEAR_JERK 50.0000,EXAX_IGN 0}
;DECL E6POS XP48={X 409.564423,Y 274.093506,Z 239.950897,A 0.0338781923,B -0.0425408930,C 179.996,S 2,T 35,E1 0.0,E2 0.0,E3 0.0,E4 0.0,E5 0.0,E6 0.0}
;DECL FDAT FP48={TOOL_NO 1,BASE_NO 0,IPO_FRAME #BASE,POINT2[] " ",TQ_STATE FALSE}
DECL PDAT PPDAT15={VEL 100.000,ACC 30.0000,APO_DIST 100.000,APO_MODE #CDIS,GEAR_JERK 50.0000,EXAX_IGN 0}
;DECL E6POS XP49={X 409.247620,Y 274.640717,Z 167.260422,A 0.0338782221,B -0.0425409339,C 179.996,S 2,T 35,E1 0.0,E2 0.0,E3 0.0,E4 0.0,E5 0.0,E6 0.0}
;DECL FDAT FP49={TOOL_NO 1,BASE_NO 0,IPO_FRAME #BASE,POINT2[] " ",TQ_STATE FALSE}
DECL LDAT LCPDAT35={VEL 2.00000,ACC 30.0000,APO_DIST 100.000,APO_FAC 50.0000,AXIS_VEL 100.000,AXIS_ACC 100.000,ORI_TYP #VAR,CIRC_TYP #BASE,JERK_FAC 50.0000,GEAR_JERK 50.0000,EXAX_IGN 0}
;DECL E6POS XP50={X 409.247620,Y 274.640717,Z 161.080627,A 0.0338782519,B -0.0425409600,C 179.996,S 2,T 35,E1 0.0,E2 0.0,E3 0.0,E4 0.0,E5 0.0,E6 0.0}
;DECL FDAT FP50={TOOL_NO 1,BASE_NO 0,IPO_FRAME #BASE,POINT2[] " ",TQ_STATE FALSE}
DECL LDAT LCPDAT36={VEL 2.00000,ACC 30.0000,APO_DIST 100.000,APO_FAC 50.0000,AXIS_VEL 100.000,AXIS_ACC 100.000,ORI_TYP #VAR,CIRC_TYP #BASE,JERK_FAC 50.0000,GEAR_JERK 50.0000,EXAX_IGN 0}
DECL GRP_TYP GGDAT10={G_APO #NO,GRP_TIME 0.700000,CTRL #OFF,DLY 0,DST 1}
;DECL E6POS XP51={X 409.239380,Y 274.640594,Z 194.437485,A 0.0345917158,B -0.0399331413,C 179.994324,S 2,T 35,E1 0.0,E2 0.0,E3 0.0,E4 0.0,E5 0.0,E6 0.0}
;DECL FDAT FP51={TOOL_NO 1,BASE_NO 0,IPO_FRAME #BASE,POINT2[] " ",TQ_STATE FALSE}
DECL LDAT LCPDAT37={VEL 2.00000,ACC 30.0000,APO_DIST 100.000,APO_FAC 50.0000,AXIS_VEL 100.000,AXIS_ACC 100.000,ORI_TYP #VAR,CIRC_TYP #BASE,JERK_FAC 50.0000,GEAR_JERK 50.0000,EXAX_IGN 0}
;DECL E6POS XP52={X 591.901306,Y 72.0268478,Z 202.051514,A 0.0345911048,B -0.0441894457,C 179.994812,S 2,T 35,E1 0.0,E2 0.0,E3 0.0,E4 0.0,E5 0.0,E6 0.0}
;DECL FDAT FP52={TOOL_NO 1,BASE_NO 0,IPO_FRAME #BASE,POINT2[] " ",TQ_STATE FALSE}
DECL LDAT LCPDAT38={VEL 2.00000,ACC 30.0000,APO_DIST 100.000,APO_FAC 50.0000,AXIS_VEL 100.000,AXIS_ACC 100.000,ORI_TYP #VAR,CIRC_TYP #BASE,JERK_FAC 50.0000,GEAR_JERK 50.0000,EXAX_IGN 0}
;DECL E6POS XP53={X 591.947388,Y 74.1291962,Z 109.399521,A 0.0345905200,B -0.0501523316,C 179.995544,S 2,T 35,E1 0.0,E2 0.0,E3 0.0,E4 0.0,E5 0.0,E6 0.0}
;DECL FDAT FP53={TOOL_NO 1,BASE_NO 0,IPO_FRAME #BASE,POINT2[] " ",TQ_STATE FALSE}
DECL LDAT LCPDAT39={VEL 2.00000,ACC 30.0000,APO_DIST 100.000,APO_FAC 50.0000,AXIS_VEL 100.000,AXIS_ACC 100.000,ORI_TYP #VAR,CIRC_TYP #BASE,JERK_FAC 50.0000,GEAR_JERK 50.0000,EXAX_IGN 0}
;DECL E6POS XP54={X 591.947388,Y 73.7645111,Z 89.2221,A 0.0345905721,B -0.0501523763,C 179.995544,S 2,T 35,E1 0.0,E2 0.0,E3 0.0,E4 0.0,E5 0.0,E6 0.0}
;DECL FDAT FP54={TOOL_NO 1,BASE_NO 0,IPO_FRAME #BASE,POINT2[] " ",TQ_STATE FALSE}
DECL LDAT LCPDAT40={VEL 2.00000,ACC 30.0000,APO_DIST 100.000,APO_FAC 50.0000,AXIS_VEL 100.000,AXIS_ACC 100.000,ORI_TYP #VAR,CIRC_TYP #BASE,JERK_FAC 50.0000,GEAR_JERK 50.0000,EXAX_IGN 0}
DECL GRP_TYP GGDAT11={G_APO #NO,GRP_TIME 0.700000,CTRL #OFF,DLY 0,DST 1}
;DECL E6POS XP55={X 591.947510,Y 73.7676544,Z 95.0133209,A 0.0351194590,B -0.0501690544,C 179.995483,S 2,T 35,E1 0.0,E2 0.0,E3 0.0,E4 0.0,E5 0.0,E6 0.0}
;DECL FDAT FP55={TOOL_NO 1,BASE_NO 0,IPO_FRAME #BASE,POINT2[] " ",TQ_STATE FALSE}
DECL LDAT LCPDAT41={VEL 2.00000,ACC 30.0000,APO_DIST 100.000,APO_FAC 50.0000,AXIS_VEL 100.000,AXIS_ACC 100.000,ORI_TYP #VAR,CIRC_TYP #BASE,JERK_FAC 50.0000,GEAR_JERK 50.0000,EXAX_IGN 0}
;DECL E6POS XP56={X 591.935547,Y 73.7661362,Z 234.094711,A 0.0351196676,B -0.0483705774,C 179.995255,S 2,T 35,E1 0.0,E2 0.0,E3 0.0,E4 0.0,E5 0.0,E6 0.0}
;DECL FDAT FP56={TOOL_NO 1,BASE_NO 0,IPO_FRAME #BASE,POINT2[] " ",TQ_STATE FALSE}
DECL LDAT LCPDAT42={VEL 2.00000,ACC 30.0000,APO_DIST 100.000,APO_FAC 50.0000,AXIS_VEL 100.000,AXIS_ACC 100.000,ORI_TYP #VAR,CIRC_TYP #BASE,JERK_FAC 50.0000,GEAR_JERK 50.0000,EXAX_IGN 0}
;DECL E6POS XP57={X 366.516113,Y 273.617981,Z 234.149399,A 0.0351134464,B -0.0560329407,C -179.998047,S 2,T 35,E1 0.0,E2 0.0,E3 0.0,E4 0.0,E5 0.0,E6 0.0}
;DECL FDAT FP57={TOOL_NO 1,BASE_NO 0,IPO_FRAME #BASE,POINT2[] " ",TQ_STATE FALSE}
DECL PDAT PPDAT16={VEL 100.000,ACC 30.0000,APO_DIST 100.000,APO_MODE #CDIS,GEAR_JERK 50.0000,EXAX_IGN 0}
;DECL E6POS XP58={X 366.253113,Y 274.323578,Z 165.167282,A 0.601378322,B -0.0560330339,C -179.998047,S 2,T 35,E1 0.0,E2 0.0,E3 0.0,E4 0.0,E5 0.0,E6 0.0}
;DECL FDAT FP58={TOOL_NO 1,BASE_NO 0,IPO_FRAME #BASE,POINT2[] " ",TQ_STATE FALSE}
DECL LDAT LCPDAT43={VEL 2.00000,ACC 30.0000,APO_DIST 100.000,APO_FAC 50.0000,AXIS_VEL 100.000,AXIS_ACC 100.000,ORI_TYP #VAR,CIRC_TYP #BASE,JERK_FAC 50.0000,GEAR_JERK 50.0000,EXAX_IGN 0}
;DECL E6POS XP59={X 367.239532,Y 274.883728,Z 165.167282,A 90.6686783,B -0.0560325347,C -179.998047,S 2,T 43,E1 0.0,E2 0.0,E3 0.0,E4 0.0,E5 0.0,E6 0.0}
;DECL FDAT FP59={TOOL_NO 1,BASE_NO 0,IPO_FRAME #BASE,POINT2[] " ",TQ_STATE FALSE}
DECL LDAT LCPDAT44={VEL 2.00000,ACC 30.0000,APO_DIST 100.000,APO_FAC 50.0000,AXIS_VEL 100.000,AXIS_ACC 100.000,ORI_TYP #VAR,CIRC_TYP #BASE,JERK_FAC 50.0000,GEAR_JERK 50.0000,EXAX_IGN 0}
DECL E6POS XP60={X 367.239532,Y 274.883728,Z 165.167282,A -0.112460792,B -0.0560319908,C -179.998047,S 2,T 35,E1 0.0,E2 0.0,E3 0.0,E4 0.0,E5 0.0,E6 0.0}
DECL FDAT FP60={TOOL_NO 1,BASE_NO 0,IPO_FRAME #BASE,POINT2[] " ",TQ_STATE FALSE}
DECL LDAT LCPDAT45={VEL 2.00000,ACC 30.0000,APO_DIST 100.000,APO_FAC 50.0000,AXIS_VEL 100.000,AXIS_ACC 100.000,ORI_TYP #VAR,CIRC_TYP #BASE,JERK_FAC 50.0000,GEAR_JERK 50.0000,EXAX_IGN 0}
DECL E6POS XP61={X 367.239532,Y 274.883728,Z 165.167282,A -42.0039558,B -0.0560317263,C -179.998047,S 2,T 35,E1 0.0,E2 0.0,E3 0.0,E4 0.0,E5 0.0,E6 0.0}
DECL FDAT FP61={TOOL_NO 1,BASE_NO 0,IPO_FRAME #BASE,POINT2[] " ",TQ_STATE FALSE}
DECL LDAT LCPDAT46={VEL 2.00000,ACC 30.0000,APO_DIST 100.000,APO_FAC 50.0000,AXIS_VEL 100.000,AXIS_ACC 100.000,ORI_TYP #VAR,CIRC_TYP #BASE,JERK_FAC 50.0000,GEAR_JERK 50.0000,EXAX_IGN 0}
DECL E6POS XP62={X 367.239532,Y 274.883728,Z 161.348145,A -42.0039558,B -0.0560317263,C -179.998047,S 2,T 35,E1 0.0,E2 0.0,E3 0.0,E4 0.0,E5 0.0,E6 0.0}
DECL FDAT FP62={TOOL_NO 1,BASE_NO 0,IPO_FRAME #BASE,POINT2[] " ",TQ_STATE FALSE}
DECL LDAT LCPDAT47={VEL 2.00000,ACC 30.0000,APO_DIST 100.000,APO_FAC 50.0000,AXIS_VEL 100.000,AXIS_ACC 100.000,ORI_TYP #VAR,CIRC_TYP #BASE,JERK_FAC 50.0000,GEAR_JERK 50.0000,EXAX_IGN 0}
DECL E6POS XP63={X 366.158112,Y 274.883728,Z 164.908157,A 0.109536953,B -0.0560314581,C -179.998047,S 2,T 35,E1 0.0,E2 0.0,E3 0.0,E4 0.0,E5 0.0,E6 0.0}
DECL FDAT FP63={TOOL_NO 1,BASE_NO 0,IPO_FRAME #BASE,POINT2[] " ",TQ_STATE FALSE}
DECL LDAT LCPDAT48={VEL 2.00000,ACC 30.0000,APO_DIST 100.000,APO_FAC 50.0000,AXIS_VEL 100.000,AXIS_ACC 100.000,ORI_TYP #VAR,CIRC_TYP #BASE,JERK_FAC 50.0000,GEAR_JERK 50.0000,EXAX_IGN 0}
DECL E6POS XP64={X 366.137909,Y 274.858826,Z 161.159546,A 0.109805077,B -0.0524299368,C 179.997955,S 2,T 35,E1 0.0,E2 0.0,E3 0.0,E4 0.0,E5 0.0,E6 0.0}
DECL FDAT FP64={TOOL_NO 1,BASE_NO 0,IPO_FRAME #BASE,POINT2[] " ",TQ_STATE FALSE}
DECL LDAT LCPDAT49={VEL 2.00000,ACC 30.0000,APO_DIST 100.000,APO_FAC 50.0000,AXIS_VEL 100.000,AXIS_ACC 100.000,ORI_TYP #VAR,CIRC_TYP #BASE,JERK_FAC 50.0000,GEAR_JERK 50.0000,EXAX_IGN 0}
DECL E6POS XP65={X 366.043427,Y 274.788635,Z 183.001053,A 0.105974533,B -0.0352026485,C 179.985397,S 2,T 35,E1 0.0,E2 0.0,E3 0.0,E4 0.0,E5 0.0,E6 0.0}
DECL FDAT FP65={TOOL_NO 1,BASE_NO 0,IPO_FRAME #BASE,POINT2[] " ",TQ_STATE FALSE}
DECL LDAT LCPDAT50={VEL 2.00000,ACC 30.0000,APO_DIST 100.000,APO_FAC 50.0000,AXIS_VEL 100.000,AXIS_ACC 100.000,ORI_TYP #VAR,CIRC_TYP #BASE,JERK_FAC 50.0000,GEAR_JERK 50.0000,EXAX_IGN 0}
DECL GRP_TYP GGDAT12={G_APO #NO,GRP_TIME 0.700000,CTRL #OFF,DLY 0,DST 1}
DECL GRP_TYP GGDAT13={G_APO #NO,GRP_TIME 0.700000,CTRL #OFF,DLY 0,DST 1}
DECL LDAT LCPDAT51={VEL 2.00000,ACC 30.0000,APO_DIST 100.000,APO_FAC 50.0000,AXIS_VEL 100.000,AXIS_ACC 100.000,ORI_TYP #VAR,CIRC_TYP #BASE,JERK_FAC 50.0000,GEAR_JERK 50.0000,EXAX_IGN 0}
DECL E6POS XP66={X 322.394409,Y 317.214203,Z 168.306381,A 0.302610844,B -0.00158163835,C 179.999359,S 2,T 35,E1 0.0,E2 0.0,E3 0.0,E4 0.0,E5 0.0,E6 0.0}
DECL FDAT FP66={TOOL_NO 1,BASE_NO 0,IPO_FRAME #BASE,POINT2[] " ",TQ_STATE FALSE}
DECL LDAT LCPDAT52={VEL 2.00000,ACC 30.0000,APO_DIST 100.000,APO_FAC 50.0000,AXIS_VEL 100.000,AXIS_ACC 100.000,ORI_TYP #VAR,CIRC_TYP #BASE,JERK_FAC 50.0000,GEAR_JERK 50.0000,EXAX_IGN 0}
DECL E6POS XP67={X 322.394409,Y 317.214203,Z 161.041107,A 0.302610904,B -0.00158164906,C 179.999359,S 2,T 35,E1 0.0,E2 0.0,E3 0.0,E4 0.0,E5 0.0,E6 0.0}
DECL FDAT FP67={TOOL_NO 1,BASE_NO 0,IPO_FRAME #BASE,POINT2[] " ",TQ_STATE FALSE}
DECL GRP_TYP GCONT={G_APO #YES,GRP_TIME 0.0,CTRL #OFF,DLY 0,DST 0}
DECL E6POS XP2={X 16.4036045,Y 13.7776031,Z 9.14540482,A 0.312648833,B -0.0643064380,C 179.960297,S 2,T 34,E1 0.0,E2 0.0,E3 0.0,E4 0.0,E5 0.0,E6 0.0}
DECL FDAT FP2={TOOL_NO 1,BASE_NO 2,IPO_FRAME #BASE,POINT2[] " ",TQ_STATE FALSE}
DECL LDAT LCPDAT53={VEL 2.00000,ACC 30.0000,APO_DIST 100.000,APO_FAC 50.0000,AXIS_VEL 100.000,AXIS_ACC 100.000,ORI_TYP #VAR,CIRC_TYP #BASE,JERK_FAC 50.0000,GEAR_JERK 50.0000,EXAX_IGN 0}
DECL E6POS XP3={X 16.3767395,Y 13.7946863,Z 40.5063667,A 0.312649697,B -0.0656919554,C 179.960114,S 2,T 34,E1 0.0,E2 0.0,E3 0.0,E4 0.0,E5 0.0,E6 0.0}
DECL FDAT FP3={TOOL_NO 1,BASE_NO 2,IPO_FRAME #BASE,POINT2[] " ",TQ_STATE FALSE}
DECL LDAT LCPDAT54={VEL 2.00000,ACC 30.0000,APO_DIST 250.000,APO_FAC 50.0000,AXIS_VEL 100.000,AXIS_ACC 100.000,ORI_TYP #VAR,CIRC_TYP #BASE,JERK_FAC 50.0000,GEAR_JERK 50.0000,EXAX_IGN 0}
DECL E6POS XP70={X 16.3767395,Y 13.7946863,Z 166.931183,A 0.312649161,B -0.0651646405,C 179.959900,S 2,T 34,E1 0.0,E2 0.0,E3 0.0,E4 0.0,E5 0.0,E6 0.0}
DECL FDAT FP70={TOOL_NO 1,BASE_NO 2,IPO_FRAME #BASE,POINT2[] " ",TQ_STATE FALSE}
DECL LDAT LCPDAT55={VEL 2.00000,ACC 30.0000,APO_DIST 250.000,APO_FAC 50.0000,AXIS_VEL 100.000,AXIS_ACC 100.000,ORI_TYP #VAR,CIRC_TYP #BASE,JERK_FAC 50.0000,GEAR_JERK 50.0000,EXAX_IGN 0}
DECL E6POS XP71={X -303.094086,Y 406.427521,Z 186.530243,A 0.312654555,B -0.0739892647,C 179.969101,S 2,T 35,E1 0.0,E2 0.0,E3 0.0,E4 0.0,E5 0.0,E6 0.0}
DECL FDAT FP71={TOOL_NO 1,BASE_NO 2,IPO_FRAME #BASE,POINT2[] " ",TQ_STATE FALSE}
DECL PDAT PPDAT17={VEL 100.000,ACC 30.0000,APO_DIST 250.000,APO_MODE #CDIS,GEAR_JERK 50.0000,EXAX_IGN 0}
DECL E6POS XP72={X 592.825500,Y -76.2150879,Z 246.850174,A 0.302610457,B 0.00424989825,C 179.994080,S 2,T 34,E1 0.0,E2 0.0,E3 0.0,E4 0.0,E5 0.0,E6 0.0}
DECL FDAT FP72={TOOL_NO 1,BASE_NO 0,IPO_FRAME #BASE,POINT2[] " ",TQ_STATE FALSE}
DECL LDAT LCPDAT56={VEL 2.00000,ACC 30.0000,APO_DIST 250.000,APO_FAC 50.0000,AXIS_VEL 100.000,AXIS_ACC 100.000,ORI_TYP #VAR,CIRC_TYP #BASE,JERK_FAC 50.0000,GEAR_JERK 50.0000,EXAX_IGN 0}
DECL E6POS XP5={X -19.4319115,Y -20.8457603,Z 118.824501,A 90.0947,B 0.0302447248,C -179.947968,S 2,T 35,E1 0.0,E2 0.0,E3 0.0,E4 0.0,E5 0.0,E6 0.0}
DECL FDAT FP5={TOOL_NO 1,BASE_NO 1,IPO_FRAME #BASE,POINT2[] " ",TQ_STATE FALSE}
DECL PDAT PPDAT18={VEL 100.000,ACC 30.0000,APO_DIST 250.000,APO_MODE #CDIS,GEAR_JERK 50.0000,EXAX_IGN 0}
DECL E6POS XP6={X -20.4997177,Y -20.8906937,Z 18.7958603,A 90.0947,B 0.0297864638,C -179.947433,S 2,T 35,E1 0.0,E2 0.0,E3 0.0,E4 0.0,E5 0.0,E6 0.0}
DECL FDAT FP6={TOOL_NO 1,BASE_NO 1,IPO_FRAME #BASE,POINT2[] " ",TQ_STATE FALSE}
DECL LDAT LCPDAT57={VEL 2.00000,ACC 30.0000,APO_DIST 250.000,APO_FAC 50.0000,AXIS_VEL 100.000,AXIS_ACC 100.000,ORI_TYP #VAR,CIRC_TYP #BASE,JERK_FAC 50.0000,GEAR_JERK 50.0000,EXAX_IGN 0}
DECL E6POS XP7={X -20.4997177,Y -20.8906918,Z 12.7720175,A 90.0947,B 0.0297864359,C -179.947433,S 2,T 35,E1 0.0,E2 0.0,E3 0.0,E4 0.0,E5 0.0,E6 0.0}
DECL FDAT FP7={TOOL_NO 1,BASE_NO 1,IPO_FRAME #BASE,POINT2[] " ",TQ_STATE FALSE}
DECL LDAT LCPDAT58={VEL 2.00000,ACC 30.0000,APO_DIST 250.000,APO_FAC 50.0000,AXIS_VEL 100.000,AXIS_ACC 100.000,ORI_TYP #VAR,CIRC_TYP #BASE,JERK_FAC 50.0000,GEAR_JERK 50.0000,EXAX_IGN 0}
DECL GRP_TYP GGDAT14={G_APO #NO,GRP_TIME 0.700000,CTRL #OFF,DLY 0,DST 1}
DECL E6POS XP8={X -20.4997177,Y -20.8906918,Z 38.0285378,A 90.0947,B 0.0297864173,C -179.947433,S 2,T 35,E1 0.0,E2 0.0,E3 0.0,E4 0.0,E5 0.0,E6 0.0}
DECL FDAT FP8={TOOL_NO 1,BASE_NO 1,IPO_FRAME #BASE,POINT2[] " ",TQ_STATE FALSE}
DECL LDAT LCPDAT59={VEL 2.00000,ACC 30.0000,APO_DIST 250.000,APO_FAC 50.0000,AXIS_VEL 100.000,AXIS_ACC 100.000,ORI_TYP #VAR,CIRC_TYP #BASE,JERK_FAC 50.0000,GEAR_JERK 50.0000,EXAX_IGN 0}
DECL E6POS XP9={X -20.5038261,Y -20.8871422,Z 117.486877,A 90.0947,B 0.0292179585,C -179.946777,S 2,T 35,E1 0.0,E2 0.0,E3 0.0,E4 0.0,E5 0.0,E6 0.0}
DECL FDAT FP9={TOOL_NO 1,BASE_NO 1,IPO_FRAME #BASE,POINT2[] " ",TQ_STATE FALSE}
DECL LDAT LCPDAT60={VEL 2.00000,ACC 30.0000,APO_DIST 250.000,APO_FAC 50.0000,AXIS_VEL 100.000,AXIS_ACC 100.000,ORI_TYP #VAR,CIRC_TYP #BASE,JERK_FAC 50.0000,GEAR_JERK 50.0000,EXAX_IGN 0}
DECL E6POS XP4={X 16.3767414,Y 13.7946863,Z 166.931183,A 0.312649161,B -0.0651646405,C 179.959900,S 2,T 34,E1 0.0,E2 0.0,E3 0.0,E4 0.0,E5 0.0,E6 0.0}
DECL FDAT FP4={TOOL_NO 1,BASE_NO 2,IPO_FRAME #BASE,POINT2[] " ",TQ_STATE FALSE}
DECL LDAT LCPDAT61={VEL 2.00000,ACC 30.0000,APO_DIST 250.000,APO_FAC 50.0000,AXIS_VEL 100.000,AXIS_ACC 100.000,ORI_TYP #VAR,CIRC_TYP #BASE,JERK_FAC 50.0000,GEAR_JERK 50.0000,EXAX_IGN 0}
DECL E6POS XP10={X 16.3586731,Y 46.4022789,Z 166.914368,A 0.312647551,B -0.0623757541,C 179.960175,S 2,T 34,E1 0.0,E2 0.0,E3 0.0,E4 0.0,E5 0.0,E6 0.0}
DECL FDAT FP10={TOOL_NO 1,BASE_NO 2,IPO_FRAME #BASE,POINT2[] " ",TQ_STATE FALSE}
DECL PDAT PPDAT19={VEL 100.000,ACC 30.0000,APO_DIST 250.000,APO_MODE #CDIS,GEAR_JERK 50.0000,EXAX_IGN 0}
DECL E6POS XP11={X 16.3767395,Y 44.2615929,Z 40.5063667,A 0.312649757,B -0.0656919703,C 179.960114,S 2,T 34,E1 0.0,E2 0.0,E3 0.0,E4 0.0,E5 0.0,E6 0.0}
DECL FDAT FP11={TOOL_NO 1,BASE_NO 2,IPO_FRAME #BASE,POINT2[] " ",TQ_STATE FALSE}
DECL LDAT LCPDAT62={VEL 2.00000,ACC 30.0000,APO_DIST 250.000,APO_FAC 50.0000,AXIS_VEL 100.000,AXIS_ACC 100.000,ORI_TYP #VAR,CIRC_TYP #BASE,JERK_FAC 50.0000,GEAR_JERK 50.0000,EXAX_IGN 0}
DECL E6POS XP12={X 16.4079704,Y 44.2029953,Z 9.14823341,A 0.312649369,B -0.0648502,C 179.960220,S 2,T 34,E1 0.0,E2 0.0,E3 0.0,E4 0.0,E5 0.0,E6 0.0}
DECL FDAT FP12={TOOL_NO 1,BASE_NO 2,IPO_FRAME #BASE,POINT2[] " ",TQ_STATE FALSE}
DECL LDAT LCPDAT63={VEL 2.00000,ACC 30.0000,APO_DIST 250.000,APO_FAC 50.0000,AXIS_VEL 100.000,AXIS_ACC 100.000,ORI_TYP #VAR,CIRC_TYP #BASE,JERK_FAC 50.0000,GEAR_JERK 50.0000,EXAX_IGN 0}
DECL E6POS XP13={X 16.4024315,Y 44.2034073,Z 34.0609856,A 0.312649041,B -0.0641606152,C 179.960281,S 2,T 34,E1 0.0,E2 0.0,E3 0.0,E4 0.0,E5 0.0,E6 0.0}
DECL FDAT FP13={TOOL_NO 1,BASE_NO 2,IPO_FRAME #BASE,POINT2[] " ",TQ_STATE FALSE}
DECL LDAT LCPDAT64={VEL 2.00000,ACC 30.0000,APO_DIST 250.000,APO_FAC 50.0000,AXIS_VEL 100.000,AXIS_ACC 100.000,ORI_TYP #VAR,CIRC_TYP #BASE,JERK_FAC 50.0000,GEAR_JERK 50.0000,EXAX_IGN 0}
DECL GRP_TYP GGDAT15={G_APO #NO,GRP_TIME 0.700000,CTRL #OFF,DLY 0,DST 1}
DECL E6POS XP14={X 16.3767414,Y 43.3087463,Z 166.931183,A 0.312649846,B -0.0656920746,C 179.960114,S 2,T 34,E1 0.0,E2 0.0,E3 0.0,E4 0.0,E5 0.0,E6 0.0}
DECL FDAT FP14={TOOL_NO 1,BASE_NO 2,IPO_FRAME #BASE,POINT2[] " ",TQ_STATE FALSE}
DECL LDAT LCPDAT65={VEL 2.00000,ACC 30.0000,APO_DIST 250.000,APO_FAC 50.0000,AXIS_VEL 100.000,AXIS_ACC 100.000,ORI_TYP #VAR,CIRC_TYP #BASE,JERK_FAC 50.0000,GEAR_JERK 50.0000,EXAX_IGN 0}
DECL E6POS XP15={X 23.0536671,Y -20.8457603,Z 118.824501,A 90.0947,B 0.0302447174,C -179.947968,S 2,T 35,E1 0.0,E2 0.0,E3 0.0,E4 0.0,E5 0.0,E6 0.0}
DECL FDAT FP15={TOOL_NO 1,BASE_NO 1,IPO_FRAME #BASE,POINT2[] " ",TQ_STATE FALSE}
DECL PDAT PPDAT20={VEL 100.000,ACC 30.0000,APO_DIST 250.000,APO_MODE #CDIS,GEAR_JERK 50.0000,EXAX_IGN 0}
DECL E6POS XP16={X 22.6327724,Y -20.8937302,Z 18.7939053,A 90.0947,B 0.0305789653,C -179.948303,S 2,T 35,E1 0.0,E2 0.0,E3 0.0,E4 0.0,E5 0.0,E6 0.0}
DECL FDAT FP16={TOOL_NO 1,BASE_NO 1,IPO_FRAME #BASE,POINT2[] " ",TQ_STATE FALSE}
DECL LDAT LCPDAT66={VEL 2.00000,ACC 30.0000,APO_DIST 250.000,APO_FAC 50.0000,AXIS_VEL 100.000,AXIS_ACC 100.000,ORI_TYP #VAR,CIRC_TYP #BASE,JERK_FAC 50.0000,GEAR_JERK 50.0000,EXAX_IGN 0}
DECL E6POS XP17={X 22.6327724,Y -20.8937302,Z 13.0147896,A 90.0947,B 0.0305789318,C -179.948303,S 2,T 35,E1 0.0,E2 0.0,E3 0.0,E4 0.0,E5 0.0,E6 0.0}
DECL FDAT FP17={TOOL_NO 1,BASE_NO 1,IPO_FRAME #BASE,POINT2[] " ",TQ_STATE FALSE}
DECL LDAT LCPDAT67={VEL 2.00000,ACC 30.0000,APO_DIST 250.000,APO_FAC 50.0000,AXIS_VEL 100.000,AXIS_ACC 100.000,ORI_TYP #VAR,CIRC_TYP #BASE,JERK_FAC 50.0000,GEAR_JERK 50.0000,EXAX_IGN 0}
DECL GRP_TYP GGDAT16={G_APO #NO,GRP_TIME 0.700000,CTRL #OFF,DLY 0,DST 1}
DECL E6POS XP87={X 22.6327724,Y -20.8937302,Z 34.0964241,A 90.0947,B 0.0305789243,C -179.948303,S 2,T 35,E1 0.0,E2 0.0,E3 0.0,E4 0.0,E5 0.0,E6 0.0}
DECL FDAT FP87={TOOL_NO 1,BASE_NO 1,IPO_FRAME #BASE,POINT2[] " ",TQ_STATE FALSE}
DECL LDAT LCPDAT68={VEL 2.00000,ACC 30.0000,APO_DIST 250.000,APO_FAC 50.0000,AXIS_VEL 100.000,AXIS_ACC 100.000,ORI_TYP #VAR,CIRC_TYP #BASE,JERK_FAC 50.0000,GEAR_JERK 50.0000,EXAX_IGN 0}
DECL LDAT LCPDAT69={VEL 2.00000,ACC 30.0000,APO_DIST 250.000,APO_FAC 50.0000,AXIS_VEL 100.000,AXIS_ACC 100.000,ORI_TYP #VAR,CIRC_TYP #BASE,JERK_FAC 50.0000,GEAR_JERK 50.0000,EXAX_IGN 0}
DECL E6POS XP18={X 22.6327724,Y -20.8937302,Z 34.0964241,A 90.0947,B 0.0305789243,C -179.948303,S 2,T 35,E1 0.0,E2 0.0,E3 0.0,E4 0.0,E5 0.0,E6 0.0}
DECL FDAT FP18={TOOL_NO 1,BASE_NO 1,IPO_FRAME #BASE,POINT2[] " ",TQ_STATE FALSE}
DECL E6POS XP19={X 22.5835114,Y -20.8997383,Z 117.474594,A 90.0947,B 0.0308456309,C -179.948410,S 2,T 35,E1 0.0,E2 0.0,E3 0.0,E4 0.0,E5 0.0,E6 0.0}
DECL FDAT FP19={TOOL_NO 1,BASE_NO 1,IPO_FRAME #BASE,POINT2[] " ",TQ_STATE FALSE}
DECL LDAT LCPDAT70={VEL 2.00000,ACC 30.0000,APO_DIST 250.000,APO_FAC 50.0000,AXIS_VEL 100.000,AXIS_ACC 100.000,ORI_TYP #VAR,CIRC_TYP #BASE,JERK_FAC 50.0000,GEAR_JERK 50.0000,EXAX_IGN 0}
DECL E6POS XP20={X 16.3551350,Y 73.3178787,Z 166.911102,A 0.312647253,B -0.0618312731,C 179.960205,S 2,T 34,E1 0.0,E2 0.0,E3 0.0,E4 0.0,E5 0.0,E6 0.0}
DECL FDAT FP20={TOOL_NO 1,BASE_NO 2,IPO_FRAME #BASE,POINT2[] " ",TQ_STATE FALSE}
DECL PDAT PPDAT21={VEL 100.000,ACC 30.0000,APO_DIST 250.000,APO_MODE #CDIS,GEAR_JERK 50.0000,EXAX_IGN 0}
DECL E6POS XP21={X 16.3767395,Y 73.8229904,Z 40.5063667,A 0.312649786,B -0.0656919777,C 179.960114,S 2,T 34,E1 0.0,E2 0.0,E3 0.0,E4 0.0,E5 0.0,E6 0.0}
DECL FDAT FP21={TOOL_NO 1,BASE_NO 2,IPO_FRAME #BASE,POINT2[] " ",TQ_STATE FALSE}
DECL LDAT LCPDAT71={VEL 2.00000,ACC 30.0000,APO_DIST 250.000,APO_FAC 50.0000,AXIS_VEL 100.000,AXIS_ACC 100.000,ORI_TYP #VAR,CIRC_TYP #BASE,JERK_FAC 50.0000,GEAR_JERK 50.0000,EXAX_IGN 0}
DECL E6POS XP22={X 16.4079704,Y 73.9751740,Z 9.14823341,A 0.312649459,B -0.0648502707,C 179.960220,S 2,T 34,E1 0.0,E2 0.0,E3 0.0,E4 0.0,E5 0.0,E6 0.0}
DECL FDAT FP22={TOOL_NO 1,BASE_NO 2,IPO_FRAME #BASE,POINT2[] " ",TQ_STATE FALSE}
DECL LDAT LCPDAT72={VEL 2.00000,ACC 30.0000,APO_DIST 250.000,APO_FAC 50.0000,AXIS_VEL 100.000,AXIS_ACC 100.000,ORI_TYP #VAR,CIRC_TYP #BASE,JERK_FAC 50.0000,GEAR_JERK 50.0000,EXAX_IGN 0}
DECL GRP_TYP GGDAT17={G_APO #NO,GRP_TIME 0.700000,CTRL #OFF,DLY 0,DST 1}
DECL E6POS XP23={X 16.4036942,Y 73.9752808,Z 35.6563263,A 0.312649131,B -0.0643085763,C 179.960236,S 2,T 34,E1 0.0,E2 0.0,E3 0.0,E4 0.0,E5 0.0,E6 0.0}
DECL FDAT FP23={TOOL_NO 1,BASE_NO 2,IPO_FRAME #BASE,POINT2[] " ",TQ_STATE FALSE}
DECL LDAT LCPDAT73={VEL 2.00000,ACC 30.0000,APO_DIST 250.000,APO_FAC 50.0000,AXIS_VEL 100.000,AXIS_ACC 100.000,ORI_TYP #VAR,CIRC_TYP #BASE,JERK_FAC 50.0000,GEAR_JERK 50.0000,EXAX_IGN 0}
DECL E6POS XP24={X 16.3767414,Y 70.8703461,Z 166.931183,A 0.312650025,B -0.0656922087,C 179.960114,S 2,T 34,E1 0.0,E2 0.0,E3 0.0,E4 0.0,E5 0.0,E6 0.0}
DECL FDAT FP24={TOOL_NO 1,BASE_NO 2,IPO_FRAME #BASE,POINT2[] " ",TQ_STATE FALSE}
DECL LDAT LCPDAT74={VEL 2.00000,ACC 30.0000,APO_DIST 250.000,APO_FAC 50.0000,AXIS_VEL 100.000,AXIS_ACC 100.000,ORI_TYP #VAR,CIRC_TYP #BASE,JERK_FAC 50.0000,GEAR_JERK 50.0000,EXAX_IGN 0}
DECL E6POS XP25={X -19.4600029,Y 22.5043011,Z 118.852913,A 90.0947,B 0.0266351383,C -179.944244,S 2,T 35,E1 0.0,E2 0.0,E3 0.0,E4 0.0,E5 0.0,E6 0.0}
DECL FDAT FP25={TOOL_NO 1,BASE_NO 1,IPO_FRAME #BASE,POINT2[] " ",TQ_STATE FALSE}
DECL PDAT PPDAT22={VEL 100.000,ACC 30.0000,APO_DIST 250.000,APO_MODE #CDIS,GEAR_JERK 50.0000,EXAX_IGN 0}
DECL E6POS XP26={X -20.5141964,Y 21.7280560,Z 18.8063393,A 90.0947,B 0.0281440206,C -179.945786,S 2,T 35,E1 0.0,E2 0.0,E3 0.0,E4 0.0,E5 0.0,E6 0.0}
DECL FDAT FP26={TOOL_NO 1,BASE_NO 1,IPO_FRAME #BASE,POINT2[] " ",TQ_STATE FALSE}
DECL LDAT LCPDAT75={VEL 2.00000,ACC 30.0000,APO_DIST 250.000,APO_FAC 50.0000,AXIS_VEL 100.000,AXIS_ACC 100.000,ORI_TYP #VAR,CIRC_TYP #BASE,JERK_FAC 50.0000,GEAR_JERK 50.0000,EXAX_IGN 0}
DECL E6POS XP27={X -20.5141964,Y 21.3681278,Z 12.6985435,A 90.0947,B 0.0281439703,C -179.945786,S 2,T 35,E1 0.0,E2 0.0,E3 0.0,E4 0.0,E5 0.0,E6 0.0}
DECL FDAT FP27={TOOL_NO 1,BASE_NO 1,IPO_FRAME #BASE,POINT2[] " ",TQ_STATE FALSE}
DECL LDAT LCPDAT76={VEL 2.00000,ACC 30.0000,APO_DIST 250.000,APO_FAC 50.0000,AXIS_VEL 100.000,AXIS_ACC 100.000,ORI_TYP #VAR,CIRC_TYP #BASE,JERK_FAC 50.0000,GEAR_JERK 50.0000,EXAX_IGN 0}
DECL GRP_TYP GGDAT18={G_APO #NO,GRP_TIME 0.700000,CTRL #OFF,DLY 0,DST 1}
DECL E6POS XP28={X -20.5096111,Y 21.3635559,Z 34.0803108,A 90.0947,B 0.0286756214,C -179.946320,S 2,T 35,E1 0.0,E2 0.0,E3 0.0,E4 0.0,E5 0.0,E6 0.0}
DECL FDAT FP28={TOOL_NO 1,BASE_NO 1,IPO_FRAME #BASE,POINT2[] " ",TQ_STATE FALSE}
DECL LDAT LCPDAT77={VEL 2.00000,ACC 30.0000,APO_DIST 250.000,APO_FAC 50.0000,AXIS_VEL 100.000,AXIS_ACC 100.000,ORI_TYP #VAR,CIRC_TYP #BASE,JERK_FAC 50.0000,GEAR_JERK 50.0000,EXAX_IGN 0}
DECL E6POS XP29={X -20.5189495,Y 20.7404461,Z 117.502289,A 90.0947,B 0.0272446107,C -179.944763,S 2,T 35,E1 0.0,E2 0.0,E3 0.0,E4 0.0,E5 0.0,E6 0.0}
DECL FDAT FP29={TOOL_NO 1,BASE_NO 1,IPO_FRAME #BASE,POINT2[] " ",TQ_STATE FALSE}
DECL LDAT LCPDAT78={VEL 2.00000,ACC 30.0000,APO_DIST 250.000,APO_FAC 50.0000,AXIS_VEL 100.000,AXIS_ACC 100.000,ORI_TYP #VAR,CIRC_TYP #BASE,JERK_FAC 50.0000,GEAR_JERK 50.0000,EXAX_IGN 0}
DECL E6POS XP30={X 16.3551350,Y 104.820755,Z 166.911102,A 0.312647253,B -0.0618313737,C 179.960205,S 2,T 35,E1 0.0,E2 0.0,E3 0.0,E4 0.0,E5 0.0,E6 0.0}
DECL FDAT FP30={TOOL_NO 1,BASE_NO 2,IPO_FRAME #BASE,POINT2[] " ",TQ_STATE FALSE}
DECL PDAT PPDAT23={VEL 100.000,ACC 30.0000,APO_DIST 250.000,APO_MODE #CDIS,GEAR_JERK 50.0000,EXAX_IGN 0}
DECL E6POS XP31={X 16.3767395,Y 104.352791,Z 40.5063667,A 0.312649786,B -0.0656919926,C 179.960114,S 2,T 35,E1 0.0,E2 0.0,E3 0.0,E4 0.0,E5 0.0,E6 0.0}
DECL FDAT FP31={TOOL_NO 1,BASE_NO 2,IPO_FRAME #BASE,POINT2[] " ",TQ_STATE FALSE}
DECL LDAT LCPDAT79={VEL 2.00000,ACC 30.0000,APO_DIST 250.000,APO_FAC 50.0000,AXIS_VEL 100.000,AXIS_ACC 100.000,ORI_TYP #VAR,CIRC_TYP #BASE,JERK_FAC 50.0000,GEAR_JERK 50.0000,EXAX_IGN 0}
DECL E6POS XP32={X 16.4079704,Y 104.088814,Z 9.14823341,A 0.312649459,B -0.0648503304,C 179.960220,S 2,T 35,E1 0.0,E2 0.0,E3 0.0,E4 0.0,E5 0.0,E6 0.0}
DECL FDAT FP32={TOOL_NO 1,BASE_NO 2,IPO_FRAME #BASE,POINT2[] " ",TQ_STATE FALSE}
DECL LDAT LCPDAT80={VEL 2.00000,ACC 30.0000,APO_DIST 250.000,APO_FAC 50.0000,AXIS_VEL 100.000,AXIS_ACC 100.000,ORI_TYP #VAR,CIRC_TYP #BASE,JERK_FAC 50.0000,GEAR_JERK 50.0000,EXAX_IGN 0}
DECL GRP_TYP GGDAT19={G_APO #NO,GRP_TIME 0.700000,CTRL #OFF,DLY 0,DST 1}
DECL E6POS XP33={X 16.3886948,Y 104.088303,Z 35.5425,A 0.312648,B -0.0624087714,C 179.960175,S 2,T 35,E1 0.0,E2 0.0,E3 0.0,E4 0.0,E5 0.0,E6 0.0}
DECL FDAT FP33={TOOL_NO 1,BASE_NO 2,IPO_FRAME #BASE,POINT2[] " ",TQ_STATE FALSE}
DECL LDAT LCPDAT81={VEL 2.00000,ACC 30.0000,APO_DIST 250.000,APO_FAC 50.0000,AXIS_VEL 100.000,AXIS_ACC 100.000,ORI_TYP #VAR,CIRC_TYP #BASE,JERK_FAC 50.0000,GEAR_JERK 50.0000,EXAX_IGN 0}
DECL E6POS XP34={X 16.3767414,Y 103.533508,Z 166.931183,A 0.312650,B -0.0656922683,C 179.960114,S 2,T 35,E1 0.0,E2 0.0,E3 0.0,E4 0.0,E5 0.0,E6 0.0}
DECL FDAT FP34={TOOL_NO 1,BASE_NO 2,IPO_FRAME #BASE,POINT2[] " ",TQ_STATE FALSE}
DECL LDAT LCPDAT82={VEL 2.00000,ACC 30.0000,APO_DIST 250.000,APO_FAC 50.0000,AXIS_VEL 100.000,AXIS_ACC 100.000,ORI_TYP #VAR,CIRC_TYP #BASE,JERK_FAC 50.0000,GEAR_JERK 50.0000,EXAX_IGN 0}
DECL E6POS XP35={X 26.3562965,Y 22.4825382,Z 118.832153,A 90.0947,B 0.0295022782,C -179.946777,S 2,T 35,E1 0.0,E2 0.0,E3 0.0,E4 0.0,E5 0.0,E6 0.0}
DECL FDAT FP35={TOOL_NO 1,BASE_NO 1,IPO_FRAME #BASE,POINT2[] " ",TQ_STATE FALSE}
DECL PDAT PPDAT24={VEL 100.000,ACC 30.0000,APO_DIST 250.000,APO_MODE #CDIS,GEAR_JERK 50.0000,EXAX_IGN 0}
DECL E6POS XP36={X 22.0406837,Y 21.7280560,Z 18.8063393,A 90.0947,B 0.0281440038,C -179.945786,S 2,T 35,E1 0.0,E2 0.0,E3 0.0,E4 0.0,E5 0.0,E6 0.0}
DECL FDAT FP36={TOOL_NO 1,BASE_NO 1,IPO_FRAME #BASE,POINT2[] " ",TQ_STATE FALSE}
DECL LDAT LCPDAT83={VEL 2.00000,ACC 30.0000,APO_DIST 250.000,APO_FAC 50.0000,AXIS_VEL 100.000,AXIS_ACC 100.000,ORI_TYP #VAR,CIRC_TYP #BASE,JERK_FAC 50.0000,GEAR_JERK 50.0000,EXAX_IGN 0}
DECL E6POS XP37={X 22.4293747,Y 21.7280579,Z 13.0520630,A 90.0947,B 0.0281439535,C -179.945786,S 2,T 35,E1 0.0,E2 0.0,E3 0.0,E4 0.0,E5 0.0,E6 0.0}
DECL FDAT FP37={TOOL_NO 1,BASE_NO 1,IPO_FRAME #BASE,POINT2[] " ",TQ_STATE FALSE}
DECL LDAT LCPDAT84={VEL 2.00000,ACC 30.0000,APO_DIST 250.000,APO_FAC 50.0000,AXIS_VEL 100.000,AXIS_ACC 100.000,ORI_TYP #VAR,CIRC_TYP #BASE,JERK_FAC 50.0000,GEAR_JERK 50.0000,EXAX_IGN 0}
DECL GRP_TYP GGDAT20={G_APO #NO,GRP_TIME 0.700000,CTRL #OFF,DLY 0,DST 1}
DECL E6POS XP38={X 22.4293747,Y 21.7280579,Z 35.4705963,A 90.0947,B 0.0281439293,C -179.945786,S 2,T 35,E1 0.0,E2 0.0,E3 0.0,E4 0.0,E5 0.0,E6 0.0}
DECL FDAT FP38={TOOL_NO 1,BASE_NO 1,IPO_FRAME #BASE,POINT2[] " ",TQ_STATE FALSE}
DECL LDAT LCPDAT85={VEL 2.00000,ACC 30.0000,APO_DIST 250.000,APO_FAC 50.0000,AXIS_VEL 100.000,AXIS_ACC 100.000,ORI_TYP #VAR,CIRC_TYP #BASE,JERK_FAC 50.0000,GEAR_JERK 50.0000,EXAX_IGN 0}
DECL E6POS XP39={X 21.6663895,Y 20.7404461,Z 117.502289,A 90.0947,B 0.0272445921,C -179.944763,S 2,T 35,E1 0.0,E2 0.0,E3 0.0,E4 0.0,E5 0.0,E6 0.0}
DECL FDAT FP39={TOOL_NO 1,BASE_NO 1,IPO_FRAME #BASE,POINT2[] " ",TQ_STATE FALSE}
DECL LDAT LCPDAT86={VEL 2.00000,ACC 30.0000,APO_DIST 250.000,APO_FAC 50.0000,AXIS_VEL 100.000,AXIS_ACC 100.000,ORI_TYP #VAR,CIRC_TYP #BASE,JERK_FAC 50.0000,GEAR_JERK 50.0000,EXAX_IGN 0}
DECL E6POS XP40={X 16.3551350,Y 137.388336,Z 166.911102,A 0.312647253,B -0.0618314072,C 179.960205,S 2,T 35,E1 0.0,E2 0.0,E3 0.0,E4 0.0,E5 0.0,E6 0.0}
DECL FDAT FP40={TOOL_NO 1,BASE_NO 2,IPO_FRAME #BASE,POINT2[] " ",TQ_STATE FALSE}
DECL PDAT PPDAT25={VEL 100.000,ACC 30.0000,APO_DIST 250.000,APO_MODE #CDIS,GEAR_JERK 50.0000,EXAX_IGN 0}
DECL E6POS XP41={X 16.3767395,Y 133.151352,Z 40.5063667,A 0.312649816,B -0.0656920299,C 179.960114,S 2,T 35,E1 0.0,E2 0.0,E3 0.0,E4 0.0,E5 0.0,E6 0.0}
DECL FDAT FP41={TOOL_NO 1,BASE_NO 2,IPO_FRAME #BASE,POINT2[] " ",TQ_STATE FALSE}
DECL LDAT LCPDAT87={VEL 2.00000,ACC 30.0000,APO_DIST 250.000,APO_FAC 50.0000,AXIS_VEL 100.000,AXIS_ACC 100.000,ORI_TYP #VAR,CIRC_TYP #BASE,JERK_FAC 50.0000,GEAR_JERK 50.0000,EXAX_IGN 0}
DECL E6POS XP42={X 16.4079704,Y 134.102188,Z 9.14823341,A 0.312649459,B -0.0648503825,C 179.960220,S 2,T 35,E1 0.0,E2 0.0,E3 0.0,E4 0.0,E5 0.0,E6 0.0}
DECL FDAT FP42={TOOL_NO 1,BASE_NO 2,IPO_FRAME #BASE,POINT2[] " ",TQ_STATE FALSE}
DECL LDAT LCPDAT88={VEL 2.00000,ACC 30.0000,APO_DIST 250.000,APO_FAC 50.0000,AXIS_VEL 100.000,AXIS_ACC 100.000,ORI_TYP #VAR,CIRC_TYP #BASE,JERK_FAC 50.0000,GEAR_JERK 50.0000,EXAX_IGN 0}
DECL GRP_TYP GGDAT21={G_APO #NO,GRP_TIME 0.700000,CTRL #OFF,DLY 0,DST 1}
DECL E6POS XP43={X 16.4079704,Y 134.102188,Z 36.9830742,A 0.312649459,B -0.0648503900,C 179.960220,S 2,T 35,E1 0.0,E2 0.0,E3 0.0,E4 0.0,E5 0.0,E6 0.0}
DECL FDAT FP43={TOOL_NO 1,BASE_NO 2,IPO_FRAME #BASE,POINT2[] " ",TQ_STATE FALSE}
DECL LDAT LCPDAT89={VEL 2.00000,ACC 30.0000,APO_DIST 250.000,APO_FAC 50.0000,AXIS_VEL 100.000,AXIS_ACC 100.000,ORI_TYP #VAR,CIRC_TYP #BASE,JERK_FAC 50.0000,GEAR_JERK 50.0000,EXAX_IGN 0}
DECL E6POS XP44={X 16.3767414,Y 132.942627,Z 166.931183,A 0.312650025,B -0.0656922907,C 179.960114,S 2,T 35,E1 0.0,E2 0.0,E3 0.0,E4 0.0,E5 0.0,E6 0.0}
DECL FDAT FP44={TOOL_NO 1,BASE_NO 2,IPO_FRAME #BASE,POINT2[] " ",TQ_STATE FALSE}
DECL LDAT LCPDAT90={VEL 2.00000,ACC 30.0000,APO_DIST 250.000,APO_FAC 50.0000,AXIS_VEL 100.000,AXIS_ACC 100.000,ORI_TYP #VAR,CIRC_TYP #BASE,JERK_FAC 50.0000,GEAR_JERK 50.0000,EXAX_IGN 0}
DECL E6POS XP45={X -19.4957752,Y 65.5391464,Z 118.893341,A 90.0946960,B 0.0212545246,C -179.939377,S 2,T 35,E1 0.0,E2 0.0,E3 0.0,E4 0.0,E5 0.0,E6 0.0}
DECL FDAT FP45={TOOL_NO 1,BASE_NO 1,IPO_FRAME #BASE,POINT2[] " ",TQ_STATE FALSE}
DECL PDAT PPDAT26={VEL 100.000,ACC 30.0000,APO_DIST 250.000,APO_MODE #CDIS,GEAR_JERK 50.0000,EXAX_IGN 0}
DECL E6POS XP46={X -20.5379219,Y 64.2026367,Z 18.8248062,A 90.0947,B 0.0252263732,C -179.943039,S 2,T 35,E1 0.0,E2 0.0,E3 0.0,E4 0.0,E5 0.0,E6 0.0}
DECL FDAT FP46={TOOL_NO 1,BASE_NO 1,IPO_FRAME #BASE,POINT2[] " ",TQ_STATE FALSE}
DECL LDAT LCPDAT91={VEL 2.00000,ACC 30.0000,APO_DIST 250.000,APO_FAC 50.0000,AXIS_VEL 100.000,AXIS_ACC 100.000,ORI_TYP #VAR,CIRC_TYP #BASE,JERK_FAC 50.0000,GEAR_JERK 50.0000,EXAX_IGN 0}
DECL E6POS XP47={X -20.5379219,Y 64.2026443,Z 12.6162472,A 90.0947,B 0.0252263471,C -179.943039,S 2,T 35,E1 0.0,E2 0.0,E3 0.0,E4 0.0,E5 0.0,E6 0.0}
DECL FDAT FP47={TOOL_NO 1,BASE_NO 1,IPO_FRAME #BASE,POINT2[] " ",TQ_STATE FALSE}
DECL LDAT LCPDAT92={VEL 2.00000,ACC 30.0000,APO_DIST 250.000,APO_FAC 50.0000,AXIS_VEL 100.000,AXIS_ACC 100.000,ORI_TYP #VAR,CIRC_TYP #BASE,JERK_FAC 50.0000,GEAR_JERK 50.0000,EXAX_IGN 0}
DECL GRP_TYP GGDAT22={G_APO #NO,GRP_TIME 0.700000,CTRL #OFF,DLY 0,DST 1}
DECL E6POS XP48={X -20.5320168,Y 64.1959534,Z 34.3267250,A 90.0947,B 0.0260242820,C -179.943741,S 2,T 35,E1 0.0,E2 0.0,E3 0.0,E4 0.0,E5 0.0,E6 0.0}
DECL FDAT FP48={TOOL_NO 1,BASE_NO 1,IPO_FRAME #BASE,POINT2[] " ",TQ_STATE FALSE}
DECL LDAT LCPDAT93={VEL 2.00000,ACC 30.0000,APO_DIST 250.000,APO_FAC 50.0000,AXIS_VEL 100.000,AXIS_ACC 100.000,ORI_TYP #VAR,CIRC_TYP #BASE,JERK_FAC 50.0000,GEAR_JERK 50.0000,EXAX_IGN 0}
DECL E6POS XP49={X -20.3022289,Y 65.1791077,Z 117.508377,A 90.0947,B 0.0263111368,C -179.944122,S 2,T 35,E1 0.0,E2 0.0,E3 0.0,E4 0.0,E5 0.0,E6 0.0}
DECL FDAT FP49={TOOL_NO 1,BASE_NO 1,IPO_FRAME #BASE,POINT2[] " ",TQ_STATE FALSE}
DECL LDAT LCPDAT94={VEL 2.00000,ACC 30.0000,APO_DIST 250.000,APO_FAC 50.0000,AXIS_VEL 100.000,AXIS_ACC 100.000,ORI_TYP #VAR,CIRC_TYP #BASE,JERK_FAC 50.0000,GEAR_JERK 50.0000,EXAX_IGN 0}
DECL E6POS XP50={X 16.3664055,Y 161.184525,Z 166.921646,A 0.312648326,B -0.0635774359,C 179.960388,S 2,T 35,E1 0.0,E2 0.0,E3 0.0,E4 0.0,E5 0.0,E6 0.0}
DECL FDAT FP50={TOOL_NO 1,BASE_NO 2,IPO_FRAME #BASE,POINT2[] " ",TQ_STATE FALSE}
DECL PDAT PPDAT27={VEL 100.000,ACC 30.0000,APO_DIST 250.000,APO_MODE #CDIS,GEAR_JERK 50.0000,EXAX_IGN 0}
DECL E6POS XP51={X 16.3767395,Y 163.818665,Z 40.5063667,A 0.312649816,B -0.0656921044,C 179.960114,S 2,T 35,E1 0.0,E2 0.0,E3 0.0,E4 0.0,E5 0.0,E6 0.0}
DECL FDAT FP51={TOOL_NO 1,BASE_NO 2,IPO_FRAME #BASE,POINT2[] " ",TQ_STATE FALSE}
DECL LDAT LCPDAT95={VEL 2.00000,ACC 30.0000,APO_DIST 250.000,APO_FAC 50.0000,AXIS_VEL 100.000,AXIS_ACC 100.000,ORI_TYP #VAR,CIRC_TYP #BASE,JERK_FAC 50.0000,GEAR_JERK 50.0000,EXAX_IGN 0}
DECL E6POS XP52={X 16.4144611,Y 164.068329,Z 9.15243530,A 0.312649965,B -0.0656600446,C 179.960312,S 2,T 35,E1 0.0,E2 0.0,E3 0.0,E4 0.0,E5 0.0,E6 0.0}
DECL FDAT FP52={TOOL_NO 1,BASE_NO 2,IPO_FRAME #BASE,POINT2[] " ",TQ_STATE FALSE}
DECL LDAT LCPDAT96={VEL 2.00000,ACC 30.0000,APO_DIST 250.000,APO_FAC 50.0000,AXIS_VEL 100.000,AXIS_ACC 100.000,ORI_TYP #VAR,CIRC_TYP #BASE,JERK_FAC 50.0000,GEAR_JERK 50.0000,EXAX_IGN 0}
DECL GRP_TYP GGDAT23={G_APO #NO,GRP_TIME 0.700000,CTRL #OFF,DLY 0,DST 1}
DECL E6POS XP53={X 16.4144611,Y 164.068329,Z 37.4588737,A 0.312649965,B -0.0656600818,C 179.960312,S 2,T 35,E1 0.0,E2 0.0,E3 0.0,E4 0.0,E5 0.0,E6 0.0}
DECL FDAT FP53={TOOL_NO 1,BASE_NO 2,IPO_FRAME #BASE,POINT2[] " ",TQ_STATE FALSE}
DECL LDAT LCPDAT97={VEL 2.00000,ACC 30.0000,APO_DIST 250.000,APO_FAC 50.0000,AXIS_VEL 100.000,AXIS_ACC 100.000,ORI_TYP #VAR,CIRC_TYP #BASE,JERK_FAC 50.0000,GEAR_JERK 50.0000,EXAX_IGN 0}
DECL E6POS XP54={X 16.3875790,Y 163.592178,Z 166.941345,A 0.312650979,B -0.0673407316,C 179.960510,S 2,T 35,E1 0.0,E2 0.0,E3 0.0,E4 0.0,E5 0.0,E6 0.0}
DECL FDAT FP54={TOOL_NO 1,BASE_NO 2,IPO_FRAME #BASE,POINT2[] " ",TQ_STATE FALSE}
DECL LDAT LCPDAT98={VEL 2.00000,ACC 30.0000,APO_DIST 250.000,APO_FAC 50.0000,AXIS_VEL 100.000,AXIS_ACC 100.000,ORI_TYP #VAR,CIRC_TYP #BASE,JERK_FAC 50.0000,GEAR_JERK 50.0000,EXAX_IGN 0}
DECL E6POS XP55={X 23.3852634,Y 65.5391464,Z 118.893341,A 90.0946960,B 0.0212544519,C -179.939377,S 2,T 43,E1 0.0,E2 0.0,E3 0.0,E4 0.0,E5 0.0,E6 0.0}
DECL FDAT FP55={TOOL_NO 1,BASE_NO 1,IPO_FRAME #BASE,POINT2[] " ",TQ_STATE FALSE}
DECL PDAT PPDAT28={VEL 100.000,ACC 30.0000,APO_DIST 250.000,APO_MODE #CDIS,GEAR_JERK 50.0000,EXAX_IGN 0}
DECL E6POS XP56={X 21.8873577,Y 64.2026367,Z 18.8248062,A 90.0947,B 0.0252263416,C -179.943039,S 2,T 43,E1 0.0,E2 0.0,E3 0.0,E4 0.0,E5 0.0,E6 0.0}
DECL FDAT FP56={TOOL_NO 1,BASE_NO 1,IPO_FRAME #BASE,POINT2[] " ",TQ_STATE FALSE}
DECL LDAT LCPDAT99={VEL 2.00000,ACC 30.0000,APO_DIST 250.000,APO_FAC 50.0000,AXIS_VEL 100.000,AXIS_ACC 100.000,ORI_TYP #VAR,CIRC_TYP #BASE,JERK_FAC 50.0000,GEAR_JERK 50.0000,EXAX_IGN 0}
DECL E6POS XP57={X 21.8873577,Y 64.2026367,Z 12.8603983,A 90.0947,B 0.0252261758,C -179.943039,S 2,T 43,E1 0.0,E2 0.0,E3 0.0,E4 0.0,E5 0.0,E6 0.0}
DECL FDAT FP57={TOOL_NO 1,BASE_NO 1,IPO_FRAME #BASE,POINT2[] " ",TQ_STATE FALSE}
DECL LDAT LCPDAT100={VEL 2.00000,ACC 30.0000,APO_DIST 250.000,APO_FAC 50.0000,AXIS_VEL 100.000,AXIS_ACC 100.000,ORI_TYP #VAR,CIRC_TYP #BASE,JERK_FAC 50.0000,GEAR_JERK 50.0000,EXAX_IGN 0}
DECL GRP_TYP GGDAT24={G_APO #NO,GRP_TIME 0.700000,CTRL #OFF,DLY 0,DST 1}
DECL E6POS XP58={X 21.8903294,Y 64.1987534,Z 35.4017639,A 90.0947,B 0.0256792,C -179.943390,S 2,T 43,E1 0.0,E2 0.0,E3 0.0,E4 0.0,E5 0.0,E6 0.0}
DECL FDAT FP58={TOOL_NO 1,BASE_NO 1,IPO_FRAME #BASE,POINT2[] " ",TQ_STATE FALSE}
DECL LDAT LCPDAT101={VEL 2.00000,ACC 30.0000,APO_DIST 250.000,APO_FAC 50.0000,AXIS_VEL 100.000,AXIS_ACC 100.000,ORI_TYP #VAR,CIRC_TYP #BASE,JERK_FAC 50.0000,GEAR_JERK 50.0000,EXAX_IGN 0}
DECL E6POS XP59={X 20.7998810,Y 65.1517563,Z 117.481819,A 90.0947,B 0.0300105885,C -179.947159,S 2,T 43,E1 0.0,E2 0.0,E3 0.0,E4 0.0,E5 0.0,E6 0.0}
DECL FDAT FP59={TOOL_NO 1,BASE_NO 1,IPO_FRAME #BASE,POINT2[] " ",TQ_STATE FALSE}
DECL LDAT LCPDAT102={VEL 2.00000,ACC 30.0000,APO_DIST 250.000,APO_FAC 50.0000,AXIS_VEL 100.000,AXIS_ACC 100.000,ORI_TYP #VAR,CIRC_TYP #BASE,JERK_FAC 50.0000,GEAR_JERK 50.0000,EXAX_IGN 0}
ENDDAT
